// Transition to the ERROR state if applicable
IF bMyMove AND stMotionStage.bError THEN
    nState := ERROR;
    bError := TRUE;
    nErrorId := stMotionStage.nErrorId;
    bCausedError := TRUE;
END_IF
sErrorMessage := F_MotionErrorCodeLookup(nErrorId := nErrorId);

CASE nState OF
INIT, WAIT_EXEC, ERROR:
    bBusy := FALSE;
ELSE
    bBusy := TRUE;
END_CASE

END_FUNCTION_BLOCK

// POUs/Motion/States/FB_PositionStateReadND
FUNCTION_BLOCK FB_PositionStateReadND
(*
    Function block to get the combined N-dimensional state of a group of motors.
    It is a building block not meant for use outside of lcls-twintcat-motion.

    Use FB_PositionStateRead1D, FB_PositionStateRead2D, ... etc. instead
*)
VAR_IN_OUT
    // The motors with a combined N-dimensional state
    astMotionStage: ARRAY[1..MotionConstants.MAX_STATE_MOTORS] OF ST_MotionStage;
    // Each motor's respective position states along its direction
    astPositionState: ARRAY[1..MotionConstants.MAX_STATE_MOTORS] OF ARRAY[1..GeneralConstants.MAX_STATES] OF ST_PositionState;
END_VAR
VAR_INPUT
    // The number of motors we're actually using
    nActiveMotorCount: UINT;
END_VAR
VAR_OUTPUT
    // TRUE if we're standing still at a known state.
    bKnownState: BOOL;
    // TRUE if we're moving, there can be no valid state if we are moving.
    bMovingState: BOOL;
    // If we're at a known state, this will be the state index along the enclosed states arrays. Otherwise, it will be zero, which is below the bounds of the states array.
    nPositionIndex: UINT;
    // TRUE if the active motor count was invalid
    bMotorCountError: BOOL;
    // A full description of whether we're at each of our states. This is used to clarify cases where states may overlap.
    abAtPosition: ARRAY[1..GeneralConstants.MAX_STATES] OF BOOL;
END_VAR
VAR
    // The individual position state reader function blocks
    afbPositionStateRead: ARRAY[1..MotionConstants.MAX_STATE_MOTORS] OF FB_PositionStateRead;

    nIter: UINT;
    nIter2: UINT;
END_VAR


CheckCount();
IF NOT bMotorCountError THEN
    DoStateReads();
    CombineOutputs();
END_IF

ACTION CheckCount:

// Make sure the motor count is valid (positive, nonzero, less or equal to the max)
bMotorCountError S= nActiveMotorCount <= 0;
bMotorCountError S= nActiveMotorCount > MotionConstants.MAX_STATE_MOTORS;
END_ACTION

ACTION CombineOutputs:

// bKnownState is TRUE if ALL motors have the same known state
bKnownState := TRUE;
FOR nIter := 1 TO nActiveMotorCount DO
    bKnownState := bKnownState AND afbPositionStateRead[nIter].bKnownState;
END_FOR

// bMovingState is TRUE if ANY motor is moving
bMovingState := FALSE;
FOR nIter := 1 TO nActiveMotorCount DO
    bMovingState := bMovingState OR afbPositionStateRead[nIter].bMovingState;
END_FOR

// To account for redundant 1D states, we need to check the full output arrays.
nPositionIndex := 0;
FOR nIter := 1 TO GeneralConstants.MAX_STATES DO
    abAtPosition[nIter] := TRUE;
    FOR nIter2 := 1 TO nActiveMotorCount DO
        abAtPosition[nIter] R= NOT afbPositionStateRead[nIter2].abAtPosition[nIter];
    END_FOR
    IF abAtPosition[nIter] THEN
        nPositionIndex := nIter;
    END_IF
END_FOR

// Position index 0 means different positions
bKnownState := bKnownState AND nPositionIndex <> 0;
END_ACTION

ACTION DoStateReads:

MOTION_GVL.nMaxStateMotorCount := MAX(MOTION_GVL.nMaxStateMotorCount, nActiveMotorCount);
FOR nIter := 1 TO nActiveMotorCount DO
    afbPositionStateRead[nIter](
        stMotionStage:=astMotionStage[nIter],
        astPositionState:=astPositionState[nIter],
    );
END_FOR
END_ACTION

END_FUNCTION_BLOCK

// POUs/Motion/States/FB_PositionStateRead
FUNCTION_BLOCK FB_PositionStateRead
(*
    This function block tells us what state a single motor is at.
    In the case of multiple valid overlapping states, one will be picked arbitrarily,
    but we can see a full description of which overlapping states are present using the abAtPosition array.

    This will only run properly if FB_PositionStateInternal has been called on each position state to initialize it.
*)
VAR_IN_OUT
    // The motor to check the state of
    stMotionStage: ST_MotionStage;
    // The allowed states for this motor
    astPositionState: ARRAY[1..GeneralConstants.MAX_STATES] OF ST_PositionState;
END_VAR
VAR_OUTPUT
    // TRUE if we're standing still at a known state, or moving within the bounds of a state to another location in the bounds.
    bKnownState: BOOL;
    // TRUE if we're moving to some other state or to another non-state position.
    bMovingState: BOOL;
    // If we're at a known state, this will be the index in the astPositionState array that matches the state. Otherwise, this will be 0, which is below the bounds of the array, so it cannot be confused with a valid output.
    nPositionIndex: UINT;
    // A copy of the details of the current position state, for convenience. This may be a moving state or an unknown state as a placeholder if we are not at a known state.
    stCurrentPosition: ST_PositionState;
    // A full description of whether we're at each of our states. This is used in 2D, 3D, etc. to clarify cases where states may overlap in 1D.
    abAtPosition: ARRAY[1..GeneralConstants.MAX_STATES] OF BOOL;
END_VAR
VAR
    nIter: UINT;
END_VAR


bKnownState := FALSE;
bMovingState := FALSE;

FOR nIter := 1 TO GeneralConstants.MAX_STATES DO
    IF astPositionState[nIter].bValid THEN
        MOTION_GVL.nMaxStates := MAX(MOTION_GVL.nMaxStates, nIter);
    END_IF
    IF F_AtPositionState(stMotionStage:=stMotionStage, stPositionState:=astPositionState[nIter]) THEN
        bKnownState := TRUE;
        nPositionIndex := nIter;
        stCurrentPosition := astPositionState[nIter];
        abAtPosition[nIter] := TRUE;
    ELSE
        abAtPosition[nIter] := FALSE;
    END_IF
END_FOR

IF NOT bKnownState THEN
    nPositionIndex := 0;
    stCurrentPosition.fPosition := stMotionStage.stAxisStatus.fActPosition;
    stCurrentPosition.fDelta := 0;
    stCurrentPosition.bMoveOk := FALSE;
    stCurrentPosition.bValid := FALSE;
    stCurrentPosition.bUseRawCounts := FALSE;

    bMovingState := stMotionStage.bExecute;
    IF bMovingState THEN
        stCurrentPosition.sName := 'Moving';
        stCurrentPosition.fVelocity := stMotionStage.fVelocity;
        stCurrentPosition.fAccel := stMotionStage.fAcceleration;
    ELSE
        stCurrentPosition.sName := 'Unknown';
    END_IF
END_IF

END_FUNCTION_BLOCK

// POUs/Deprecated/FB_PositionStateManager
{attribute 'obsolete' := 'Use FB_PositionState1D instead'}
FUNCTION_BLOCK FB_PositionStateManager
(*
    Handles EPICS moves between multiple states for a single axis
    Should be wrapped inside a block with enums for states,
    see FB_EpicsInOut for an example.
*)
VAR_IN_OUT
    // Motor to move
    stMotionStage: ST_MotionStage;

    // Allocated space for 15 states besides Unknown (16 is the max for an EPICS MBBI)
    {attribute 'pytmc' := '
        pv:
        io: io
        expand: %.2d
    '}
    arrStates: ARRAY[1..15] OF ST_PositionState;

    // Corresponding arrStates index to move to, or 0 if no move selected
    setState: INT;
END_VAR
VAR_INPUT
    // If TRUE, start a move when setState transitions to a nonzero number
    bEnable: BOOL;
    // On rising edge, reset this FB
    {attribute 'pytmc' := '
        pv: RESET
        io: io
        field: ZNAM False
        field: ONAM True
    '}
    bReset: BOOL;
END_VAR
VAR_OUTPUT
    // If TRUE, there is an error
    {attribute 'pytmc' := '
        pv: ERR
        io: i
        field: ZNAM False
        field: ONAM True
    '}
    bError: BOOL;
    // Error ID
    {attribute 'pytmc' := '
        pv: ERRID
        io: i
    '}
    nErrorId: UDINT;
    // The error that caused bError to flip TRUE
    {attribute 'pytmc' := '
        pv: ERRMSG
        io: i
    '}
    sErrorMessage: STRING;
    // If TRUE, we are moving the motor
    {attribute 'pytmc' := '
        pv: BUSY
        io: i
        field: ZNAM False
        field: ONAM True
    '}
    bBusy: BOOL;
    // If TRUE, we are not moving the motor and the last move completed successfully
    {attribute 'pytmc' := '
        pv: DONE
        io: i
        field: ZNAM False
        field: ONAM True
    '}
    bDone: BOOL;

    // The current position we are trying to reach, or 0
    goalState: INT;
    // The readback position
    getState: INT;
END_VAR
VAR
    bInit: BOOL;
    stUnknown: ST_PositionState;
    stGoal: ST_PositionState;
    fbStateMove: FB_PositionStateMove;
    fbStateInternal: ARRAY[1..15] OF FB_PositionStateInternal;
    nIndex: INT;
    bNewGoal: BOOL;
    bInnerExec: BOOL;
    bInnerReset: BOOL;
    rtReset: R_TRIG;
    bMoveRequested: BOOL;
END_VAR

// Reset just goes through the first-cycle init again
rtReset(CLK:=bReset);
IF rtReset.Q THEN
    bInit := FALSE;
END_IF

// First-cycle init
IF NOT bInit THEN
    bError := FALSE;
    sErrorMessage := '';
    bBusy := FALSE;
    bDone := FALSE;
    bNewGoal := FALSE;
    bInnerExec := FALSE;
    bInnerReset := TRUE;
    setState := 0;
    goalState := 0;
END_IF

// All state internal handlers
FOR nIndex := 1 TO 15 DO
    IF arrStates[nIndex].bValid THEN
        fbStateInternal[nIndex](
            stMotionStage:=stMotionStage,
            stPositionState:=arrStates[nIndex]);
    END_IF
END_FOR

// Check where we are by going through all possible states.
// Note this favors the highest-number state that we're at, it's up to you to make your states mutually exclusive.
getState := 0;
FOR nIndex := 1 TO 15 DO
    IF F_AtPositionState(stMotionStage:=stMotionStage, stPositionState:=arrStates[nIndex]) THEN
        getState := nIndex;
    END_IF
END_FOR

// Use the changing set pv as a rising-edge trigger
IF setState <> goalState THEN
    goalState := setState;
    bNewGoal := TRUE;
END_IF

// Special move handling for error/enable state
IF bError OR NOT bEnable THEN
    bInnerExec := FALSE;
// Reset inner block this cycle if we were already moving but want a new move
ELSIF bInnerExec AND bNewGoal THEN
    bInnerExec := FALSE;
    bInnerReset := TRUE;
// If we hit this branch, we're starting a new move
ELSIF bNewGoal THEN
    bInnerExec := TRUE;
    bInnerReset := FALSE;
    bNewGoal := FALSE;
END_IF

// Pick the correct goal structure or Unknown
IF goalState = 0 THEN
    stGoal := stUnknown;
ELSE
    stGoal := arrStates[goalState];
END_IF

// Do the move
fbStateMove(
    stMotionStage := stMotionStage,
    stPositionState := stGoal,
    bExecute := bInnerExec,
    bReset := bInnerReset,
    enumMotionRequest := E_MotionRequest.INTERRUPT,
    bBusy => bBusy);

// Only pass up bDone information if this FB is active
IF bInnerExec THEN
    bDone := fbStateMove.bDone;
END_IF

// Pick up any new errors, but don't override uncleared existing errors
IF NOT bError THEN
    bError := fbStateMove.bError;
    nErrorId := fbStateMove.nErrorId;
    sErrorMessage := fbStateMove.sErrorMessage;
END_IF

// Reset the setpoint and goal to 0 if we're not doing anything
// because FB is waiting for a change from 0 to "something"
bMoveRequested := bInnerExec AND NOT bDone;
IF NOT bError AND NOT bNewGoal AND NOT bMoveRequested THEN
    setState := 0;
    goalState := 0;
    bInnerExec := FALSE;
END_IF

// Bring inner reset back low at the end of the init cycle so that it can be triggered again later
IF NOT bInit THEN
    bInit := TRUE;
    bInnerReset := FALSE;
END_IF

END_FUNCTION_BLOCK

// POUs/Deprecated/FB_PositionStateBase
{attribute 'obsolete' := 'Use FB_PositionState1D instead'}
FUNCTION_BLOCK FB_PositionStateBase
(*
    Handles EPICS moves between multiple states for a single axis
    Should be subclassed for a specific enumSet and enumGet.
    See body comment  or FB_PositionStateInOut for an implementation example.
*)
VAR_IN_OUT
    // Motor to move
    stMotionStage: ST_MotionStage;
END_VAR
VAR_INPUT
    // If TRUE, start a move when setState transitions to a nonzero number
    bEnable: BOOL;
    // On rising edge, reset this FB
    {attribute 'pytmc' := '
        pv: RESET
        io: io
        field: ZNAM False
        field: ONAM True
    '}
    bReset: BOOL;
END_VAR
VAR_OUTPUT
    // If TRUE, there is an error
    {attribute 'pytmc' := '
        pv: ERR
        io: i
        field: ZNAM False
        field: ONAM True
    '}
    bError: BOOL;
    // Error ID
    {attribute 'pytmc' := '
        pv: ERRID
        io: i
    '}
    nErrorId: UDINT;
    // The error that caused bError to flip TRUE
    {attribute 'pytmc' := '
        pv: ERRMSG
        io: i
    '}
    sErrorMessage: STRING;
    // If TRUE, we are moving the motor
    {attribute 'pytmc' := '
        pv: BUSY
        io: i
        field: ZNAM False
        field: ONAM True
    '}
    bBusy: BOOL;
    // If TRUE, we are not moving the motor and the last move completed successfully
    {attribute 'pytmc' := '
        pv: DONE
        io: i
        field: ZNAM False
        field: ONAM True
    '}
    bDone: BOOL;
END_VAR
VAR
    // Pre-allocated array of states
    {attribute 'pytmc' := '
        pv:
        io: io
        expand: %.2d
    '}
    arrStates: ARRAY[1..GeneralConstants.MAX_STATES] OF ST_PositionState;

    // Corresponding arrStates index to move to, or 0 if no move selected
    setState: INT;
    // The current position we are trying to reach, or 0
    goalState: INT;
    // The readback position
    getState: INT;

    bInit: BOOL;
    stUnknown: ST_PositionState;
    stGoal: ST_PositionState;
    fbStateMove: FB_PositionStateMove;
    fbStateInternal: ARRAY[1..GeneralConstants.MAX_STATES] OF FB_PositionStateInternal;
    nIndex: INT;
    bNewGoal: BOOL;
    bInnerExec: BOOL;
    bInnerReset: BOOL;
    rtReset: R_TRIG;
    bMoveRequested: BOOL;
END_VAR

(*
    Subclass me, define enums to translate setState and getState, call Exec

    Example:

    <something to fill arrStates>
    setState := enumSet;
    Exec();
    enumGet := getState;
    enumSet := setState;
*)

ACTION Exec:
StateHandler();
END_ACTION

ACTION StateHandler:
// Reset just goes through the first-cycle init again
rtReset(CLK:=bReset);
IF rtReset.Q THEN
    bInit := FALSE;
    bReset := FALSE;
END_IF

// First-cycle init
IF NOT bInit THEN
    bError := FALSE;
    nErrorID := 0;
    sErrorMessage := '';
    bBusy := FALSE;
    bDone := FALSE;
    bNewGoal := FALSE;
    bInnerExec := FALSE;
    bInnerReset := TRUE;
    setState := 0;
    goalState := 0;
END_IF

// All state internal handlers
FOR nIndex := 1 TO GeneralConstants.MAX_STATES DO
    IF arrStates[nIndex].bValid THEN
        fbStateInternal[nIndex](
            stMotionStage:=stMotionStage,
            stPositionState:=arrStates[nIndex]);
    END_IF
END_FOR

// Check where we are by going through all possible states.
// Note this favors the highest-number state that we're at, it's up to you to make your states mutually exclusive.
getState := 0;
FOR nIndex := 1 TO GeneralConstants.MAX_STATES DO
    IF F_AtPositionState(stMotionStage:=stMotionStage, stPositionState:=arrStates[nIndex]) THEN
        getState := nIndex;
    END_IF
END_FOR

// Use the changing set pv as a rising-edge trigger
IF setState <> goalState THEN
    goalState := setState;
    bNewGoal := TRUE;
END_IF

// Special move handling for error/enable state
IF bError OR NOT bEnable THEN
    bInnerExec := FALSE;
ELSIF bNewGoal THEN
    IF fbStateMove.bBusy THEN
        // Stop previous move if we were already moving but want a new move
        bInnerExec := FALSE;
    ELSE
        // If we hit this branch, we're ready to start a new move
        bInnerExec := TRUE;
        bInnerReset := FALSE;
        bNewGoal := FALSE;
    END_IF
END_IF

// Pick the correct goal structure or Unknown
IF goalState = 0 THEN
    stGoal := stUnknown;
ELSE
    stGoal := arrStates[goalState];
END_IF

// Do the move
fbStateMove(
    stMotionStage := stMotionStage,
    stPositionState := stGoal,
    bExecute := bInnerExec,
    bReset := bInnerReset,
    enumMotionRequest := E_MotionRequest.INTERRUPT,
    bBusy => bBusy);

// Only pass up bDone information if this FB is active
IF bInnerExec THEN
    bDone := fbStateMove.bDone;
END_IF

// Pick up any new errors, but don't override uncleared existing errors
IF NOT bError THEN
    bError := fbStateMove.bError;
    IF bError THEN
        nErrorId := fbStateMove.nErrorId;
        sErrorMessage := fbStateMove.sErrorMessage;
    END_IF
END_IF

// Reset the setpoint and goal to 0 if we're not doing anything
// because FB is waiting for a change from 0 to "something"
bMoveRequested := bInnerExec AND NOT bDone;
IF NOT bError AND NOT bNewGoal AND NOT bMoveRequested THEN
    setState := 0;
    goalState := 0;
    bInnerExec := FALSE;
END_IF

// Bring inner reset back low at the end of the init cycle so that it can be triggered again later
IF NOT bInit THEN
    bInit := TRUE;
    bInnerReset := FALSE;
END_IF
END_ACTION

END_FUNCTION_BLOCK

// POUs/Deprecated/FB_PositionStateInOut
{attribute 'obsolete' := 'Use FB_PositionState1D_InOut instead'}
FUNCTION_BLOCK FB_PositionStateInOut EXTENDS FB_PositionStateBase
(*
    Example usage of FB_PositionStateBase for a simple IN/OUT axis. See NOTE: comments.
    Also usable as a drop-in for these cases (no need to roll your own in/out)
*)
VAR_INPUT
    // The enum position to move to
    {attribute 'pytmc' := '
        pv: SET
        io: io
    '}
    enumSet: ENUM_EpicsInOut_INT; // NOTE: Please copy this pragma exactly on your enumSet

    // Information about the OUT position
    stOut: ST_PositionState; // NOTE: Do not pragma these, let it happen in the manager.
    // Information about the IN position
    stIn: ST_PositionState;
END_VAR
VAR_OUTPUT
    // The enum state readback
    {attribute 'pytmc' := '
        pv: GET
        io: i
    '}
    enumGet: ENUM_EpicsInOut_INT; // NOTE: Please copy this pragma exactly on your enumGet
END_VAR
VAR
    bInOutInit: BOOL;
END_VAR

IF NOT bInOutInit THEN
    bInOutInit := TRUE;
    arrStates[1] := stOut;
    arrStates[2] := stIn;
    stOut.sName := 'OUT';
    stIn.sName := 'IN';
END_IF
setState := enumSet;
Exec();
enumGet := getState;
enumSet := setState;

END_FUNCTION_BLOCK

// POUs/Deprecated/FB_PositionStateBase_WithPMPS
{attribute 'obsolete' := 'Use FB_PositionStatePMPS1D instead'}
FUNCTION_BLOCK FB_PositionStateBase_WithPMPS EXTENDS FB_PositionStateBase
(*
    Handles EPICS moves between multiple states for a single axis with PMPS.
    Should be subclassed for a specific enumSet and enumGet.
    See body comment  or FB_PositionStateInOut_WithPMPS for an implementation example.
*)
VAR_IN_OUT
    fbArbiter: FB_Arbiter;
    fbFFHWO: FB_HardwareFFOutput;
END_VAR
VAR_INPUT
    sPmpsDeviceName: STRING;
    sTransitionKey: STRING;
    {attribute 'pytmc' := '
        pv: PMPS:ARB:ENABLE
        io: io
    '}
    bArbiterEnabled: BOOL := TRUE;
    tArbiterTimeout: TIME := T#1s;
    bMoveOnArbiterTimeout: BOOL := TRUE;
    fStateBoundaryDeadband: LREAL := 0;
    bBPOKAutoReset: BOOL := False;
END_VAR
VAR
    {attribute 'pytmc' := 'pv: PMPS'}
    fbStatePMPS: FB_PositionStatePMPS;
    fbEncErrFFO: FB_EncErrorFFO;
END_VAR

(*
    Subclass me, define enums to translate setState and getState, call Exec

    Example:

    <something to fill arrStates>
    setState := enumSet;
    Exec();
    enumGet := getState;
    enumSet := setState;
*)

ACTION Exec:
StateHandler();
PMPSHandler();
END_ACTION

ACTION PMPSHandler:
fbStatePMPS(
    fbArbiter:=fbArbiter,
    fbFFHWO:=fbFFHWO,
    stMotionStage:=stMotionStage,
    arrStates:=arrStates,
    sPmpsDeviceName:=sPmpsDeviceName,
    sTransitionKey:=sTransitionKey,
    stPmpsDoc:= PMPS_GVL.BP_jsonDoc,
    bRequestTransition:=setState <> 0,
    setState:=setState,
    getState:=getState,
    bArbiterEnabled:=bArbiterEnabled,
    tArbiterTimeout:=tArbiterTimeout,
    bMoveOnArbiterTimeout:=bMoveOnArbiterTimeout,
    fStateBoundaryDeadband:=fStateBoundaryDeadband,
    bBPOKAutoReset:=bBPOKAutoReset);

fbEncErrFFO(
    stMotionStage:=stMotionStage,
    fbFFHWO:=fbFFHWO,
    bAutoReset:=TRUE);
END_ACTION

END_FUNCTION_BLOCK

// POUs/Deprecated/FB_PositionStateInOut_WithPMPS
{attribute 'obsolete' := 'Use FB_PositionStatePMPS1D_InOut instead'}
FUNCTION_BLOCK FB_PositionStateInOut_WithPMPS EXTENDS FB_PositionStateBase_WithPMPS
(*
    Example usage of FB_PositionStateBase_WithPMPS for a simple IN/OUT axis. See NOTE: comments.
    Also usable as a drop-in for these cases (no need to roll your own in/out)

    This is the PMPS version. Note that the only difference is that we extend the _WithPMPS FB.
*)
VAR_INPUT
    // The enum position to move to
    {attribute 'pytmc' := '
        pv: SET
        io: io
    '}
    enumSet: ENUM_EpicsInOut_INT; // NOTE: Please copy this pragma exactly on your enumSet

    // Information about the OUT position
    stOut: ST_PositionState; // NOTE: Do not pragma these, let it happen in the manager.
    // Information about the IN position
    stIn: ST_PositionState;
END_VAR
VAR_OUTPUT
    // The enum state readback
    {attribute 'pytmc' := '
        pv: GET
        io: i
    '}
    enumGet: ENUM_EpicsInOut_INT; // NOTE: Please copy this pragma exactly on your enumGet
END_VAR
VAR
    bInOutInit: BOOL;
END_VAR

IF NOT bInOutInit THEN
    bInOutInit := TRUE;
    arrStates[1] := stOut;
    arrStates[2] := stIn;
    stOut.sName := 'OUT';
    stIn.sName := 'IN';
END_IF
setState := enumSet;
Exec();
enumGet := getState;
enumSet := setState;

END_FUNCTION_BLOCK

// POUs/Motion/States/Examples/FB_PositionStatePMPS1D_InOut
FUNCTION_BLOCK FB_PositionStatePMPS1D_InOut
(*
    An example and usable drop-in instance for a 1D pmps state device with just an IN and an OUT state.
    Note that the outward-facing API is nearly identical to the non-PMPS version
*)
VAR_IN_OUT
    // Include a stage that can be passed into the FB
    stMotionStage: ST_MotionStage;
    // Simplify the interface, the user just needs to construct and pass in and out position states
    stIn: ST_PositionState;
    stOut: ST_PositionState;
    // Include PMPS output helpers
    fbFFHWO: FB_HardwareFFOutput;
    fbArbiter: FB_Arbiter;
END_VAR
VAR_INPUT
    // Define an ENUM for EPICS to use to set a new value. It is expected this will be written to during one cycle, so don't continually apply a value here in the PLC code.
    // It is exposed as an input so we can test it using the PLC.
    {attribute 'pytmc' := '
      pv: STATE:SET
      io: io
    '}
    eStateSet: E_EpicsInOut;
END_VAR
VAR_OUTPUT
    // Define an ENUM for EPICS to use to report the new value.
    {attribute 'pytmc' := '
      pv: STATE:GET
      io: i
    '}
    eStateGet: E_EpicsInOut;
END_VAR
VAR
    // Include the standard fb with blank pv pragma
    {attribute 'pytmc' := 'pv:'}
    fbPositionStatePMPS1D: FB_PositionStatePMPS1D;
    // The standard fb expects a full array of position states
    astPositionState: ARRAY[1..GeneralConstants.MAX_STATES] OF ST_PositionState;
END_VAR


// Optional: default state names
IF stIn.sName = '' THEN
    stIn.sName := 'IN';
END_IF
IF stOut.sName = '' THEN
    stOut.sName := 'OUT';
END_IF

// Assemble the states array, matching the enum values
astPositionState[E_EpicsInOut.OUT] := stOut;
astPositionState[E_EpicsInOut.IN] := stIn;

// Call the main function block, passing our motors, states, and an enable
fbPositionStatePMPS1D(
    fbFFHWO:=fbFFHWO,
    fbArbiter:=fbArbiter,
    stMotionStage:=stMotionStage,
    astPositionState:=astPositionState,
    eEnumSet:=eStateSet,
    eEnumGet:=eStateGet,
    bEnableMotion:=TRUE,
    bEnableBeamParams:=TRUE,
    bEnablePositionLimits:=TRUE,
);

// Send updates made on the array back to the inputs (VAR_IN_OUT) for maximum clarity
stOut := astPositionState[E_EpicsInOut.OUT];
stIn := astPositionState[E_EpicsInOut.IN];

END_FUNCTION_BLOCK

// POUs/Deprecated/FB_PositionStatePMPS
{attribute 'obsolete' := 'Use FB_PositionStatePMPS1D instead'}
FUNCTION_BLOCK FB_PositionStatePMPS EXTENDS FB_PositionStatePMPS_Base
(*
    Hooks up a position state to an arbiter and an FFO
        Use BeamParameterTransitionManager to manage transition requests between states
        Hook up to the inputs/outputs of the state function block
        Raises FFO if beam parameters are worse than required for current state
*)
VAR_IN_OUT
    fbArbiter: FB_Arbiter;
    fbFFHWO: FB_HardwareFFOutput;
END_VAR
VAR_INPUT
    bReadPmpsDb: BOOL;
    sPmpsDeviceName: STRING;
    sTransitionKey: STRING;
    stPmpsDoc: SJsonValue;
    stHighBeamThreshold: ST_BeamParams := PMPS_GVL.cstFullBeam;
    bBPOKAutoReset: BOOL := False;
END_VAR
VAR
    arrPMPS: ARRAY[0..GeneralConstants.MAX_STATES] OF ST_DbStateParams;
    nBPIndex: UINT;
    nTransitionAssertionID: UDINT;
    nLastReqAssertionID: UDINT;
    fbReadPmpsDb: FB_JsonDocToSafeBP;
    ftDbBusy: F_TRIG;
    rtReadDBExec: R_TRIG;
    ftRead: F_TRIG;
    bptm: BeamParameterTransitionManager;
    ffBeamParamsOk: FB_FastFault;
    ffZeroRate: FB_FastFault;
    ffBPTMTimeoutAndMove: FB_FastFault;
    ffBPTMError: FB_FastFault;
    ffMaint: FB_FastFault;
    ffUnknown: FB_FastFault;
    bFFOxOk: BOOL;
    bAtSafeState: BOOL;
    nIter: UINT;
END_VAR

Exec();

ACTION AssertHere:
fbArbiter.AddRequest(
    sDevName := stMotionStage.sName,
    nReqID := stStateReq.stPMPS.nRequestAssertionID,
    stReqBP := stStateReq.stPMPS.stBeamParams);
END_ACTION

ACTION ClearAsserts:
fbArbiter.RemoveRequest(nTransitionAssertionID);
FOR nIter := 1 TO GeneralConstants.MAX_STATES DO
    fbArbiter.RemoveRequest(arrStates[nIter].stPMPS.nRequestAssertionID);
END_FOR
END_ACTION

ACTION HandleBPTM:
(*
  Handle finishing the bptm late if timed out
  bptm needs a rising edge of bTransDone after authorizing transition
  If we fall into this block, bTransDone would otherwise be stuck at TRUE forever
  so the BPTM would never see a rising edge and therefore stay stuck
  We set to FALSE here to reset the BPTM, then gets set to TRUE again if really done.
*)
rtDoLateFinish(CLK:=bLateFinish AND bInternalAuth);
IF rtDoLateFinish.Q THEN
    bTransDone := FALSE;
    bLateFinish := FALSE;
END_IF

IF stStateReq.stPMPS.nRequestAssertionID <> nTransitionAssertionID THEN
    (*
        Edge case: the request is swapped out without a move
        Same as above: we need a rising edge of bTransDone, so cause a falling edge and the let the rising edge happen next cycle
        This will already be false when we request a positional move
    *)
    bTransDone R= stStateReq.stPMPS.nRequestAssertionID <> nLastReqAssertionID;
    // Just normal bptm call
    bptm(fbArbiter:=fbArbiter,
         i_sDeviceName:=stMotionStage.sName,
         i_TransitionAssertionID:=nTransitionAssertionID,
         i_stTransitionAssertion:=stTransitionBeam,
         i_nRequestedAssertionID:=stStateReq.stPMPS.nRequestAssertionID,
         i_stRequestedAssertion:=stStateReq.stPMPS.stBeamParams,
         i_xDoneMoving:=bTransDone,
         stCurrentBeamParameters:=PMPS_GVL.stCurrentBeamParameters,
         q_xTransitionAuthorized=>bInternalAuth,
         bDone=>bBPTMDone);
    nLastReqAssertionID := stStateReq.stPMPS.nRequestAssertionID;
END_IF
END_ACTION

ACTION HandleFFO:
// stBeamNeeded will point to Unknown/No beam if we are out of state bounds or in motion
// Otherwise we'll have the current state's beam parameters

// Check for bad conditions
bFFOxOk := F_SafeBPCompare(PMPS_GVL.stCurrentBeamParameters, stBeamNeeded);
// It is safe to reset automatically if our current state can take full beam.
// Otherwise we'll have to ask for a user acknowledgement to clear.
// This avoids rapidly cycling the FFOs on/off
// You can pass in a different stHighBeamThreshold as an input parameter to customize this behavior
bAtSafeState := F_SafeBPCompare(stHighBeamThreshold, stBeamNeeded);

// If the beam parameters are wrong, it is a fault! This encompasses all unknown arbiter-related errors.
ffBeamParamsOk.i_xOK := bFFOxOk;
ffBeamParamsOk.i_xReset S= bFFOxOk AND bAtSafeState;
ffBeamParamsOk.i_xReset R= NOT ffBeamParamsOk.i_xOK;
ffBeamParamsOk.i_xAutoReset := bBPOKAutoReset;

ffBeamParamsOk(
    i_DevName:=stMotionStage.sName,
    i_Desc:='Beam parameter mismatch',
    i_TypeCode:=16#1000,
    io_fbFFHWO:=fbFFHWO);

// Trip the beam for zero-rate states. This is a PMPS training wheel and should ultimately be removed.
// Note: I think this is already redundant
ffZeroRate(
    i_xOk := stBeamNeeded.nRate > 0,
    i_xAutoReset := TRUE,
    i_DevName := stMotionStage.sName,
    i_Desc := 'Device requesting zero rate',
    i_TypeCode := 16#1001,
    io_fbFFHWO := fbFFHWO);

// Trip the beam for BPTM timeouts if we want to move
// Only reset at safe beam OR at no bptm errors (some other FF should catch additional issues)
ffBPTMTimeoutAndMove.i_xOK := NOT (bArbiterTimeout AND bMoveOnArbiterTimeout);
ffBPTMTimeoutAndMove.i_xReset S= bAtSafeState OR (bptm.bDone AND NOT bptm.bError);
ffBPTMTimeoutAndMove.i_xReset R= NOT ffBPTMTimeoutAndMove.i_xOK;
ffBPTMTimeoutAndMove(
    i_DevName := stMotionStage.sName,
    i_Desc := 'BPTM Timeout',
    i_TypeCode := 16#1002,
    io_fbFFHWO := fbFFHWO);

// Trip the beam for BPTM Errors
ffBPTMError.i_xOK := NOT bptm.bError;
ffBPTMError.i_xReset S= bptm.bDone AND NOT bptm.bError;
ffBPTMError.i_xReset R= NOT ffBPTMError.i_xOK;
ffBPTMError(
    i_DevName := stMotionStage.sName,
    i_Desc := 'BPTM error, state transition failed',
    i_TypeCode := 16#1003,
    io_fbFFHWO := fbFFHWO);

// Trip the beam for maintenance mode
ffMaint(
    i_xOK := NOT bMaintMode,
    i_xAutoReset := TRUE,
    i_DevName := stMotionStage.sName,
    i_Desc := 'Device is in maintenance mode',
    i_TypeCode := 16#1004,
    io_fbFFHWO := fbFFHWO);

// Trip the beam for unknown state
ffUnknown(
    i_xOK := getState > 0 OR bInTransition,
    i_xAutoReset := TRUE,
    i_DevName := stMotionStage.sName,
    i_Desc := 'Unknown position between moves',
    i_TypeCode := 16#1005,
    io_fbFFHWO := fbFFHWO);
END_ACTION

ACTION HandlePmpsDb:

// Automatically read from the pmps db when it updates
// Assume update if no longer busy and no errors

ftDbBusy(CLK:=MOTION_GVL.fbPmpsFileReader.bBusy);
IF ftDbBusy.Q THEN
    bReadPmpsDb S= NOT MOTION_GVL.fbPmpsFileReader.bError;
END_IF

rtReadDBExec(CLK:=bReadPmpsDb);
IF rtReadDBExec.Q THEN
    arrPMPS[0].sPmpsState := sTransitionKey;
    FOR nBPIndex := 1 TO GeneralConstants.MAX_STATES BY 1 DO
        arrPMPS[nBPIndex] := arrStates[nBPIndex].stPMPS;
    END_FOR
END_IF

fbReadPmpsDb(
    bExecute:=bReadPmpsDb,
    jsonDoc:=stPmpsDoc,
    sDeviceName:=sPmpsDeviceName,
    io_fbFFHWO:=fbFFHWO,
    arrStates:=arrPMPS,
);
bReadPmpsDb R= NOT fbReadPmpsDb.bBusy;

ftRead(CLK:=fbReadPmpsDb.bBusy);

stTransitionState.sName := 'Transition';
IF ftRead.Q AND NOT fbReadPmpsDb.bError THEN
    stTransitionDb := arrPMPS[0];
    stTransitionBeam := arrPMPS[0].stBeamParams;
    nTransitionAssertionID := arrPMPS[0].nRequestAssertionID;
    stTransitionState.stPMPS := arrPMPS[0];
    FOR nBPIndex := 1 TO GeneralConstants.MAX_STATES BY 1 DO
        arrStates[nBPIndex].stPMPS := arrPMPS[nBPIndex];
    END_FOR
END_IF
END_ACTION

END_FUNCTION_BLOCK

// POUs/Deprecated/FB_PositionStatePMPS_Base
{attribute 'obsolete' := 'Use FB_PositionStatePMPS1D instead'}
FUNCTION_BLOCK FB_PositionStatePMPS_Base
(*
    FB_PositionStatePMPS without Arbiter, BPTM, FFO

    This allows me to test most of the code without an arbiter plc setup
*)
VAR_IN_OUT
    stMotionStage: ST_MotionStage;
    arrStates: ARRAY[1..GeneralConstants.MAX_STATES] OF ST_PositionState;
END_VAR
VAR_INPUT
    bArbiterEnabled: BOOL := TRUE;
    {attribute 'pytmc' := '
        pv: MAINT
        io: io
    '}
    bMaintMode: BOOL;
    bRequestTransition: BOOL;
    setState: INT;
    getState: INT;
    fStateBoundaryDeadband: LREAL := 0;
    tArbiterTimeout: TIME := T#1s;
    bMoveOnArbiterTimeout: BOOL := TRUE;
END_VAR
VAR_OUTPUT
    bTransitionAuthorized: BOOL;
    bForwardAuthorized: BOOL;
    bBackwardAuthorized: BOOL;
    bArbiterTimeout: BOOL;
END_VAR
VAR
    {attribute 'pytmc' := '
        pv: TRANS
        io: i
    '}
    stTransitionDb: ST_DbStateParams;
    stTransitionBeam: ST_BeamParams := PMPS_GVL.cst0RateBeam;
    stTransitionState: ST_PositionState;
    bInit: BOOL := TRUE;
    bTransDone: BOOL;
    rtTransReq: R_TRIG;
    bBPTMDone: BOOL;
    rtBPTMDone: R_TRIG;
    ftMotorExec: F_TRIG;
    rtTransDone: R_TRIG;
    rtDoLateFinish: R_TRIG;
    tonDone: TON;
    stStateReq: ST_PositionState;
    mcPower: MC_POWER;
    fUpperBound: LREAL;
    fLowerBound: LREAL;
    nGoalState: INT;
    stGoalState: ST_PositionState;
    fActPos: LREAL;
    fReqPos: LREAL;
    bInTransition: BOOL;
    stBeamNeeded: ST_BeamParams;
    bFwdOk: BOOL;
    bBwdOk: BOOL;
    tonArbiter: TON;
    bLateFinish: BOOL;
    bInternalAuth: BOOL;
END_VAR

// This is meant to be subclassed. The parent class body is in the Exec action.

ACTION AssertHere:

END_ACTION

ACTION ClearAsserts:

END_ACTION

ACTION Exec:

// Load the pmps parameters as needed
HandlePmpsDb();

// Initialize or reinitialize to the current state value
rtBPTMDone(CLK:=bBPTMDone);
ftMotorExec(CLK:=stMotionStage.bExecute);
tonDone(
    IN:=bTransDone,
    PT:=T#100ms
    );
IF rtBPTMDone.Q OR ftMotorExec.Q OR tonDone.Q THEN
    bInit := TRUE;
END_IF
IF bInit OR nGoalState = 0 OR stMotionStage.bError THEN
    bInit R= stMotionStage.bAxisParamsInit;
    nGoalState := getState;
    stStateReq := GetStateStruct(getState);
    bInTransition := FALSE;
    rtTransReq(CLK:=FALSE);
    bTransitionAuthorized := FALSE;
    bArbiterTimeout := FALSE;
END_IF

// Request transition on rising edge
rtTransReq(CLK:=bRequestTransition);
IF rtTransReq.Q THEN
    nGoalState := setState;
    stStateReq := GetStateStruct(setState);
    bInTransition := TRUE;
    bTransDone := FALSE;
ELSE
    bTransDone := F_AtPositionState(stMotionStage:=stMotionStage, stPositionState:=stStateReq) AND NOT stMotionStage.bBusy;
END_IF

// Mark late finish if bTransDone -> true before the bptm is done
// This means that we finished the move so fast that the bptm needs to be unstuck via toggling bTransDone
rtTransDone(CLK:=bTransDone);
bLateFinish S= rtTransDone.Q AND NOT bBPTMDone;

IF bArbiterEnabled THEN
    // Handles getting the request to the arbiter and back
    HandleBPTM();
    // Handle arbiter timeouts
    IF tArbiterTimeout > T#0s THEN
        tonArbiter(
            IN:=bInTransition AND NOT bInternalAuth,
            PT:=tArbiterTimeout,
            Q=>bArbiterTimeout);
    ELSE
        bArbiterTimeout := FALSE;
    END_IF
    bTransitionAuthorized S= bInternalAuth OR (bArbiterTimeout AND bMoveOnArbiterTimeout);
ELSE
    // Clear all of our assertions if we decide to disable the arbiter
    ClearAsserts();
    // Do some dummy request handling
    bTransitionAuthorized := stMotionStage.bExecute;
    bArbiterTimeout := stMotionStage.bExecute;
END_IF

// Set up MPS virtual limit for moves at and between states
stGoalState := GetStateStruct(nGoalState);
fActPos := stMotionStage.stAxisStatus.fActPosition;
IF stMotionStage.bExecute THEN
    fReqPos := stMotionStage.fPosition;
ELSE
    fReqPos := fActPos;
END_IF

// Start with no move authority
bForwardAuthorized := FALSE;
bBackwardAuthorized := FALSE;

// Check if it would be OK to move without granting auth
bFwdOk := F_PosUnderUpperBound(MAX(fActPos, fReqPos) + ABS(fStateBoundaryDeadband), stGoalState);
bBwdOk := F_PosOverLowerBound(MIN(fActPos, fReqPos) - ABS(fStateBoundaryDeadband), stGoalState);

// Grant auth during moves based on goal state, current position, and goal position
IF stMotionStage.bExecute AND stGoalState.bValid THEN
    bForwardAuthorized := bFwdOk;
    bBackwardAuthorized := bBwdOk;
END_IF

IF bInTransition THEN
    // Deny auth during a transition request until transition is authorized
    bForwardAuthorized R= NOT bTransitionAuthorized;
    bBackwardAuthorized R= NOT bTransitionAuthorized;
    // Have the motor wait for permission to start move instead of immediately erroring
    stMotionStage.bSafetyReady := bTransitionAuthorized;
ELSE
    // If not transitioning, no need to wait for safety: immediately try to move and error if no auth
    stMotionStage.bSafetyReady := stMotionStage.bExecute;
    // Set an error message override in case this causes an error
    IF stMotionStage.bError AND bArbiterEnabled AND NOT bMaintMode THEN
        IF fReqPos > fActPos AND NOT bFwdOk THEN
            stMotionStage.sCustomErrorMessage := 'Unsafe tweak forward blocked by PMPS';
        ELSIF fReqPos < fActPos AND NOT bBwdOk THEN
            stMotionStage.sCustomErrorMessage := 'Unsafe tweak backward blocked by PMPS';
        END_IF
    END_IF
END_IF

IF bArbiterEnabled AND NOT bMaintMode THEN
// Only let us move if the transition is allowed, or if we are moving within a state's bounds
    mcPower(Axis:=stMotionStage.Axis,
            Enable:=stMotionStage.bAllEnable,
            Enable_Positive:=stMotionStage.bAllForwardEnable AND bForwardAuthorized,
            Enable_Negative:=stMotionStage.bAllBackwardEnable AND bBackwardAuthorized);
ELSE
    mcPower(Axis:=stMotionStage.Axis,
            Enable:=stMotionStage.bAllEnable,
            Enable_Positive:=stMotionStage.bAllForwardEnable,
            Enable_Negative:=stMotionStage.bAllBackwardEnable);
    stMotionStage.bSafetyReady := TRUE;
END_IF

// Raise fast faults as needed
stBeamNeeded := GetBeamFromState(getState);
HandleFFO();
END_ACTION

METHOD GetBeamFromState : ST_BeamParams;
VAR_INPUT
    nState: INT;
END_VAR
VAR
    stState: ST_PositionState;
END_VAR
stState := GetStateStruct(nState);
GetBeamFromState := stState.stPMPS.stBeamParams;
END_METHOD

METHOD GetStateCode : INT
VAR_INPUT
    nState: INT;
END_VAR
IF nState < 0 OR nState > GeneralConstants.MAX_STATES THEN
    GetStateCode := -1;
ELSE
    GetStateCode := nState;
END_IF
END_METHOD

METHOD GetStateStruct : ST_PositionState
VAR_INPUT
    nState: INT;
END_VAR
{warning disable C0371}
// Implicit VAR_IN_OUT reference inside a method needs special handling
IF NOT __ISVALIDREF(arrStates) THEN
    GetStateStruct := stTransitionState;
    RETURN;
END_IF
CASE GetStateCode(nState) OF
    -1: GetStateStruct := stTransitionState;
    0: GetStateStruct := stTransitionState;
    ELSE
        GetStateStruct := arrStates[nState];
END_CASE
{warning restore C0371}
END_METHOD

ACTION HandleBPTM:

END_ACTION

ACTION HandleFFO:

END_ACTION

ACTION HandlePmpsDb:

END_ACTION

END_FUNCTION_BLOCK

// POUs/Deprecated/FB_PositionStateBase_WithPMPS_Test
{attribute 'obsolete' := 'No longer any reason to use this, all state classes can have unit tests.'}
FUNCTION_BLOCK FB_PositionStateBase_WithPMPS_Test EXTENDS FB_PositionStateBase
(*
    Handles EPICS moves between multiple states for a single axis with fake PMPS.
    Should be subclassed for a specific enumSet and enumGet.
    See body comment  or FB_PositionStateInOut_WithPMPS_Test for an implementation example.
*)
VAR_INPUT
    stTransitionBeam: ST_BeamParams := PMPS_GVL.cst0RateBeam;
    nTransitionAssertionID: UDINT;
END_VAR
VAR
    fbStatePMPS: FB_PositionStatePMPS_Test;
END_VAR

(*
    Subclass me, define enums to translate setState and getState, call Exec

    Example:

    <something to fill arrStates>
    setState := enumSet;
    Exec();
    enumGet := getState;
    enumSet := setState;
*)

ACTION Exec:
StateHandler();
PMPSHandler();
END_ACTION

ACTION PMPSHandler:
fbStatePMPS(
    stMotionStage:=stMotionStage,
    arrStates:=arrStates,
    bRequestTransition:=setState <> 0,
    setState:=setState,
    getState:=getState);
END_ACTION

END_FUNCTION_BLOCK

// POUs/Deprecated/FB_PositionStateInOut_WithPMPS_Test
{attribute 'obsolete' := 'No longer any reason to use this, all state classes can have unit tests.'}
FUNCTION_BLOCK FB_PositionStateInOut_WithPMPS_Test EXTENDS FB_PositionStateBase_WithPMPS_Test
(*
    Example usage of FB_PositionStateBase_WithPMPS_Test for a simple IN/OUT axis. See NOTE: comments.
    Also usable as a drop-in for these cases (no need to roll your own in/out)

    This is the PMPS version. Note that the only difference is that we extend the _WithPMPS_Test FB.
*)
VAR_INPUT
    // The enum position to move to
    {attribute 'pytmc' := '
        pv: SET
        io: io
    '}
    enumSet: ENUM_EpicsInOut_INT; // NOTE: Please copy this pragma exactly on your enumSet

    // Information about the OUT position
    stOut: ST_PositionState; // NOTE: Do not pragma these, let it happen in the manager.
    // Information about the IN position
    stIn: ST_PositionState;
END_VAR
VAR_OUTPUT
    // The enum state readback
    {attribute 'pytmc' := '
        pv: GET
        io: i
    '}
    enumGet: ENUM_EpicsInOut_INT; // NOTE: Please copy this pragma exactly on your enumGet
END_VAR
VAR
    bInOutInit: BOOL;
END_VAR

IF NOT bInOutInit THEN
    bInOutInit := TRUE;
    arrStates[1] := stOut;
    arrStates[2] := stIn;
    stOut.sName := 'OUT';
    stIn.sName := 'IN';
END_IF
setState := enumSet;
Exec();
enumGet := getState;
enumSet := setState;

END_FUNCTION_BLOCK

// POUs/Deprecated/FB_PositionStatePMPS_Test
{attribute 'obsolete' := 'No longer any reason to use this, all state classes can have unit tests.'}
FUNCTION_BLOCK FB_PositionStatePMPS_Test EXTENDS FB_PositionStatePMPS_Base
(*
    Implement position state pmps with no FFO and auto-accept transition after 3s
    Use for offline testing of everything except the explicit interface
*)
VAR
    tonReq: TON;
END_VAR

Exec();

ACTION HandleBPTM:
// Send the fake BPTM our assertion request by changing stStateReq.stBeamParams
// We expect to recieve bTransitionAuthorized TRUE after some delta T
// We expect bTransitionAuthorized to go FALSE after stMotionStage.bBusy goes FALSE
tonReq(
    IN:=bInTransition,
    PT:=T#3s);
bTransitionAuthorized := tonReq.Q AND stMotionStage.bExecute;
END_ACTION

ACTION HandleFFO:
// Skip implementing this for offline testing
// We won't be able to tell if it worked anyway
END_ACTION

END_FUNCTION_BLOCK

// POUs/Deprecated/FB_StatePTPMove
{attribute 'obsolete' := 'Use FB_PositionStateMove instead'}
FUNCTION_BLOCK FB_StatePTPMove
// Do not use, this is deprecated
VAR_INPUT
    {attribute 'pytmc' := '
        pv:
    '}
    stPositionState: ST_PositionState;

    {attribute 'pytmc' := '
        pv: GO
        io: io
        field: ZNAM False
        field: ONAM True
    '}
    bExecute: BOOL;

    bMoveOk: BOOL;
END_VAR
VAR_IN_OUT
    stMotionStage: ST_MotionStage;
END_VAR
VAR_OUTPUT
    {attribute 'pytmc' := '
        pv: AT_STATE
        io: input
        field: ZNAM False
        field: ONAM True
    '}
    bAtState: BOOL;

    {attribute 'pytmc' := '
        pv: DMOV
        io: input
        field: ZNAM False
        field: ONAM True
    '}
    bDone: BOOL;

    {attribute 'pytmc' := '
        pv: BUSY
        io: input
        field: ZNAM False
        field: ONAM True
    '}
    bBusy: BOOL;

    {attribute 'pytmc' := '
        pv: ERR
        io: input
        field: ZNAM False
        field: ONAM True
    '}
    bError: BOOL;

    {attribute 'pytmc' := '
        pv: ERRMSG
        io: input
    '}
    sError: STRING;
END_VAR
VAR
    bExecTrig: R_TRIG;
    bExecEnd: F_TRIG;
    fActPosition: LREAL;
    fLowPos: LREAL;
    fHighPos: LREAL;
END_VAR

bExecTrig(CLK:=bExecute);
IF bExecTrig.Q AND bMoveOk THEN
    IF NOT stMotionStage.bBusy AND NOT stMotionStage.bError THEN
        stMotionStage.bExecute := TRUE;
        stMotionStage.nCommand := E_EpicsMotorCmd.MOVE_ABSOLUTE;
        stMotionStage.fPosition := stPositionState.fPosition;
        stMotionStage.fVelocity := stPositionState.fVelocity;
        stMotionStage.fAcceleration := stPositionState.fAccel;
        stMotionStage.fDeceleration := stPositionState.fDecel;
        bDone := FALSE;
        bBusy := TRUE;
    END_IF
END_IF
bError := stMotionStage.bError;
sError := stMotionStage.sErrorMessage;

fActPosition := stMotionStage.stAxisStatus.fActPosition;
fLowPos := stPositionState.fPosition - stPositionState.fDelta;
fHighPos := stPositionState.fPosition + stPositionState.fDelta;
IF (fLowPos < fActPosition) AND (fHighPos > fActPosition) THEN
    bAtState := TRUE;
    IF NOT stMotionStage.bBusy THEN
        bDone := TRUE;
        bBusy := FALSE;
        bExecute := FALSE;
    END_IF
ELSE
    bAtState := FALSE;
END_IF

bExecEnd(CLK:=bExecute);
IF bExecEnd.Q AND bBusy THEN
    stMotionStage.bExecute := FALSE;
END_IF

IF NOT stMotionStage.bExecute OR NOT bExecute THEN
    bDone := TRUE;
    bBusy := FALSE;
    bExecute := FALSE;
END_IF

END_FUNCTION_BLOCK

// POUs/ImplicitChecks/CheckBounds
// Implicitly generated code : DO NOT EDIT
FUNCTION CheckBounds : DINT
VAR_INPUT
    index, lower, upper: DINT;
END_VAR

// Implicitly generated code : Only an Implementation suggestion
{noflow}
IF  index < lower THEN
    CheckBounds := lower;
ELSIF  index > upper THEN
    CheckBounds := upper;
ELSE
    CheckBounds := index;
END_IF
{flow}

END_FUNCTION

// POUs/ImplicitChecks/CheckDivDInt
// Implicitly generated code : DO NOT EDIT
FUNCTION CheckDivDInt : DINT
VAR_INPUT
    divisor:DINT;
END_VAR

// Implicitly generated code : Only an Implementation suggestion
{noflow}
IF divisor = 0 THEN
    CheckDivDInt:=1;
ELSE
    CheckDivDInt:=divisor;
END_IF;
{flow}

END_FUNCTION

// POUs/ImplicitChecks/CheckDivLInt
// Implicitly generated code : DO NOT EDIT
FUNCTION CheckDivLInt : LINT
VAR_INPUT
    divisor:LINT;
END_VAR

// Implicitly generated code : Only an Implementation suggestion
{noflow}
IF divisor = 0 THEN
    CheckDivLInt:=1;
ELSE
    CheckDivLInt:=divisor;
END_IF;
{flow}

END_FUNCTION

// POUs/ImplicitChecks/CheckDivLReal
// Implicitly generated code : DO NOT EDIT
FUNCTION CheckDivLReal : LREAL
VAR_INPUT
    divisor:LREAL;
END_VAR

// Implicitly generated code : Only an Implementation suggestion
{noflow}
IF divisor = 0 THEN
    CheckDivLReal:=1;
ELSE
    CheckDivLReal:=divisor;
END_IF;
{flow}

END_FUNCTION

// POUs/ImplicitChecks/CheckDivReal
// Implicitly generated code : DO NOT EDIT
FUNCTION CheckDivReal : REAL
VAR_INPUT
    divisor:REAL;
END_VAR

// Implicitly generated code : Only an Implementation suggestion
{noflow}
IF divisor = 0 THEN
    CheckDivReal:=1;
ELSE
    CheckDivReal:=divisor;
END_IF;
{flow}

END_FUNCTION

// POUs/Motion/Gantry/FB_GantryAutoCoupling
FUNCTION_BLOCK FB_GantryAutoCoupling
VAR_INPUT
    nGantryTol : LINT;
END_VAR
VAR_OUTPUT
    bGantryAlreadyCoupled : BOOL;
END_VAR
VAR_IN_OUT
    Master : ST_MotionStage;
    MasterEnc : ST_RenishawAbsEnc;
    Slave : ST_MotionStage;
    SlaveEnc : ST_RenishawAbsEnc;
    bExecuteCouple : BOOL;
    bExecuteDecouple : BOOL;
END_VAR
VAR
    gantry_diff_limit : FB_GantryDiffVirtualLimitSwitch;
    couple : MC_GEARIN;
    decouple : MC_GEAROUT;
    bInitComplete : BOOL;
    fbSetEnables : FB_SetEnables;
END_VAR

// Designate Master and SLave Axes
Master.bGantryAxis := TRUE;
Slave.bGantryAxis := TRUE;

Master.nGantryTol := nGantryTol;
Slave.nGantryTol := Master.nGantryTol;

// Activate Gantry Virtual Limit Switch
gantry_diff_limit(Penc:=MasterEnc, SEnc:=SlaveEnc, GantDiffTol:=Master.nGantryTol,
                  PLimFwd=>Master.bGantryForwardEnable, PLimBwd=>Master.bGantryBackwardEnable,
                  SLimFwd=>Slave.bGantryForwardEnable, SLimBwd=>Slave.bGantryBackwardEnable);

// Coupling Status Bit
bGantryAlreadyCoupled := Master.Axis.NcToPlc.CoupleState=1 AND Slave.Axis.NcToPlc.CoupleState=3;

fbSetEnables(stMotionStage:=Master);
fbSetEnables(stMotionStage:=Slave);

IF bGantryAlreadyCoupled THEN
    Master.bGantryForwardEnable := Master.bGantryForwardEnable AND Slave.bAllForwardEnable;
    Slave.bGantryForwardEnable := Master.bAllForwardEnable AND Slave.bGantryForwardEnable;

    Master.bGantryBackwardEnable := Master.bGantryBackwardEnable AND Slave.bAllBackwardEnable;
    Slave.bGantryBackwardEnable := Master.bAllBackwardEnable AND Slave.bGantryBackwardEnable;
END_IF


// Coupling states
// Auto-coupling at init and auto-reset of coupling boolean
bExecuteCouple S= NOT bInitComplete;

bExecuteCouple R= couple.Busy OR bGantryAlreadyCoupled;
couple(Master:=Master.Axis, Slave:=Slave.Axis, Execute:=bExecuteCouple);

bInitComplete S= bGantryAlreadyCoupled;

// Decoupling with auto-reset of coupling boolean
bExecuteDecouple R= decouple.Busy OR NOT bGantryAlreadyCoupled;
decouple(Slave:=Slave.Axis, Execute:=bExecuteDecouple);

END_FUNCTION_BLOCK

// POUs/Motion/Gantry/FB_GantryDiffVirtualLimitSwitch
FUNCTION_BLOCK FB_GantryDiffVirtualLimitSwitch
VAR_INPUT
    PEnc: ST_RenishawAbsEnc; // Primary axis encoder (usually the upstream one)
    SEnc: ST_RenishawAbsEnc; // Secondary axis encoder (couples to the primary)

    GantDiffTol: LINT;        // Gantry differenace tolerance in encoder counts
END_VAR
VAR_OUTPUT
    PLimFwd: BOOL; // Primary axis forward direction enable
    PLimBwd: BOOL; // Primary axis reverse direction enable
    SLimFwd: BOOL; // Secondary axis forward direction enable
    SLimBwd: BOOL; // Secondary axis reverse direction enable
END_VAR
VAR
    GantryDiff: LINT;
END_VAR

(* Gantry Difference Virtual Limit Switch
A. Wallace 2017-2-15

Determines which direction is disabled due to it increasing the gantry difference.
Refer to the ESD for actual conventions.

A positive gantry error refers to a CCW clocked assembly:
eg. for X
X1 upstream, X2 downstream. Primary axis is always upstream.
Gantry difference > 0 when
X2>X1
Therefore
X2 positive direction disabled
X1 negative direction disabled

Call before FB_MotionStage fb calls for the gantry axes.
*)

GantryDiff := ( ULINT_TO_LINT(PEnc.Count) - ULINT_TO_LINT(PEnc.Ref) ) - ( ULINT_TO_LINT(SEnc.Count) - ULINT_TO_LINT(SEnc.Ref) );

IF ABS(GantryDiff) > GantDiffTol THEN
    IF GantryDiff < 0  THEN
        PLimBwd := FALSE;
        SLimFwd := FALSE;
    ELSE
        PLimBwd := TRUE;
        SLimFwd := TRUE;
    END_IF
    IF GantryDiff > 0 THEN
        PLimFwd := FALSE;
        SLimBwd := FALSE;
    ELSE
        PLimFwd := TRUE;
        SLimBwd := TRUE;
    END_IF
ELSE
    //If there is no fault, all directions are enabled
    PLimFwd := TRUE;
    PLimBwd := TRUE;
    SLimFwd := TRUE;
    SLimBwd := TRUE;
END_IF

END_FUNCTION_BLOCK

// POUs/Motion/PMPS/FB_PositionStatePMPS3D
FUNCTION_BLOCK FB_PositionStatePMPS3D
(*
    3-Dimensional position state function block with PMPS.

    This allows the user to move 3 motors among some set of named state positions with PMPS protection.

    To use a states block, you must define enums that match the state options and give them pytmc pragmas.
    See FB_PositionState1D_InOut for a simple example.
    These enums must be passed in as the eEnumSet and eEnumGet VAR_IN_OUT variables.
    The enum values must match the array indices in astPositionState1, astPositionState2, and astPositionState3.

    A move will begin when eEnumSet is set to a positive, nonzero value. eEnumSet will be reset to 0 on every cycle, allowing us
    to accept a new, possibly conflicting, move request on the next cycle to interrupt the first.

    The motors must already be set up for point-to-point motion via FB_MotionStage, etc., for this function block to work properly.

    PMPS handling is done via database lookups by setting sPmpsState on each position state and on
    the transition state input appropriately.
*)
VAR_IN_OUT
    // The 1st motor to move
    stMotionStage1: ST_MotionStage;
    // The 2nd motor to move
    stMotionStage2: ST_MotionStage;
    // The 3rd motor to move
    stMotionStage3: ST_MotionStage;
    // All possible position states for motor 1, including unused/invalid states.
    {attribute 'pytmc' := '
        pv: STATE:M1
        io: io
        expand: :%.2d
    '}
    astPositionState1: ARRAY[1..GeneralConstants.MAX_STATES] OF ST_PositionState;
    // All possible position states for motor 2, including unused/invalid states.
    {attribute 'pytmc' := '
        pv: STATE:M2
        io: io
        expand: :%.2d
    '}
    astPositionState2: ARRAY[1..GeneralConstants.MAX_STATES] OF ST_PositionState;
    // All possible position states for motor 3, including unused/invalid states.
    {attribute 'pytmc' := '
        pv: STATE:M3
        io: io
        expand: :%.2d
    '}
    astPositionState3: ARRAY[1..GeneralConstants.MAX_STATES] OF ST_PositionState;
    // Set this to a nonzero value to request a new move. It will be reset to zero every cycle. This should be hooked up to a user's EPICS enum input.
    eEnumSet: UINT;
    // The current state index, or zero if we are not at a state. This should be hooked up to a user's EPICS enum output.
    eEnumGet: UINT;
    // The fast fault output to fault to.
    fbFFHWO: FB_HardwareFFOutput;
    // The arbiter to request beam conditions from.
    fbArbiter: FB_Arbiter;
END_VAR
VAR_INPUT
    // Set this to TRUE to enable input state moves, or FALSE to disable them.
    bEnableMotion: BOOL;
    // Set this to TRUE to enable beam parameter checks, or FALSE to disable them.
    bEnableBeamParams: BOOL;
    // Set this to TRUE to enable position limit checks, or FALSE to disable them.
    bEnablePositionLimits: BOOL;
    // The name of the device for use in the PMPS DB lookup and diagnostic screens.
    sDeviceName: STRING;
    // The name of the transition state in the PMPS database.
    sTransitionKey: STRING;
    // Normal EPICS inputs, gathered into a single struct
    {attribute 'pytmc' := 'pv: STATE'}
    // PMPS EPICS inputs, gathered into a single struct
    stEpicsToPlc: ST_StateEpicsToPlc;
    {attribute 'pytmc' := 'pv: STATE'}
    stPMPSEpicsToPlc: ST_StatePMPSEpicsToPlc;
    // Set this to TRUE to re-read the loaded database immediately (useful for debug)
    bReadDBNow: BOOL;
END_VAR
VAR_OUTPUT
    // Normal EPICS outputs, gathered into a single struct
    {attribute 'pytmc' := 'pv: STATE'}
    stPlcToEpics: ST_StatePlcToEpics;
    // PMPS EPICS outputs, gathered into a single struct
    {attribute 'pytmc' := 'pv: STATE'}
    stPMPSPlcToEpics: ST_StatePMPSPlcToEpics;
    // The PMPS database lookup associated with the current position state.
    stDbStateParams: ST_DbStateParams;
END_VAR
VAR
    fbCore: FB_PositionStateND_Core;
    fbPMPSCore: FB_PositionStatePMPSND_Core;
    astMotionStageMax: ARRAY[1..MotionConstants.MAX_STATE_MOTORS] OF ST_MotionStage;
    astPositionStateMax: ARRAY[1..MotionConstants.MAX_STATE_MOTORS] OF ARRAY[1..GeneralConstants.MAX_STATES] OF ST_PositionState;
END_VAR


astMotionStageMax[1] := stMotionStage1;
astMotionStageMax[2] := stMotionStage2;
astMotionStageMax[3] := stMotionStage3;
astPositionStateMax[1] := astPositionState1;
astPositionStateMax[2] := astPositionState2;
astPositionStateMax[3] := astPositionState3;

fbCore(
    astMotionStageMax:=astMotionStageMax,
    astPositionStateMax:=astPositionStateMax,
    stEpicsToPlc:=stEpicsToPlc,
    stPlcToEpics:=stPlcToEpics,
    eEnumSet:=eEnumSet,
    eEnumGet:=eEnumGet,
    bEnable:=bEnableMotion,
    nActiveMotorCount:=3,
    nCurrGoal=>,
);
fbPMPSCore(
    astMotionStageMax:=astMotionStageMax,
    astPositionStateMax:=astPositionStateMax,
    stEpicsToPlc:=stEpicsToPlc,
    stPMPSEpicsToPlc:=stPMPSEpicsToPlc,
    stPlcToEpics:=stPlcToEpics,
    stPMPSPlcToEpics:=stPMPSPlcToEpics,
    fbFFHWO:=fbFFHWO,
    fbArbiter:=fbArbiter,
    bEnableBeamParams:=bEnableBeamParams,
    bEnablePositionLimits:=bEnablePositionLimits,
    nActiveMotorCount:=3,
    sDeviceName:=sDeviceName,
    sTransitionKey:=sTransitionKey,
    nCurrGoal:=fbCore.nCurrGoal,
    bReadDBNow:=bReadDBNow,
    stDbStateParams=>stDbStateParams,
);

stMotionStage1 := astMotionStageMax[1];
stMotionStage2 := astMotionStageMax[2];
stMotionStage3 := astMotionStageMax[3];
astPositionState1 := astPositionStateMax[1];
astPositionState2 := astPositionStateMax[2];
astPositionState3 := astPositionStateMax[3];

END_FUNCTION_BLOCK

// POUs/Motion/PMPS/FB_Standard_PMPSDB
FUNCTION_BLOCK FB_Standard_PMPSDB
(*
    This FB should be run on every motion PLC to encapsulate the pmps file reader.
    It is pre-instantiated at MOTION_GVL.fbStandardPMPSDB
*)
VAR_IN_OUT
    // The fast fault output to fault to.
    io_fbFFHWO: FB_HardwareFFOutput;
END_VAR
VAR_INPUT
    // If TRUE, FB will run. Reads when enable goes TRUE.
    bEnable: BOOL;
    // E.g. lfe-motion
    sPlcName: STRING;
    {attribute 'pytmc' := '
        pv: REFRESH
        io: io
    '}
    // Set to TRUE to cause an extra read.
    bRefresh: BOOL;
    // Directory where the DB is stored.
    sDirectory: STRING := '';
END_VAR
VAR_OUTPUT
    {attribute 'pytmc' := '
        pv: LAST_REFRESH
        io: i
    '}
    nLastRefreshTime: DINT;
    bReadPmpsDb: BOOL;
END_VAR
VAR
    bExecute: BOOL;
    rtEnable: R_TRIG;
    rtRefresh: R_TRIG;
    ftBusy: F_TRIG;

    // Time tracking liften from Arbiter PLCs
    fbTime : FB_LocalSystemTime := ( bEnable := TRUE, dwCycle := 1 );
    fbTime_to_UTC: FB_TzSpecificLocalTimeToSystemTime;
    fbGetTimeZone: FB_GetTimeZoneInformation;

    fbIPCReg: FB_IPCDiag_Register;
    fbCheckOS: FB_IPCDiag_ReadParameter;
    sOSName: STRING := '';
    nCheckOSTries: UINT := 3;
END_VAR

IF NOT bEnable THEN
    RETURN;
END_IF

rtEnable(CLK:=bEnable);
rtRefresh(CLK:=bRefresh);
bRefresh := FALSE;

IF rtEnable.Q OR rtRefresh.Q THEN
    // Make sure file reader gets a rising edge
    MOTION_GVL.fbPmpsFileReader(
        io_fbFFHWO:=io_fbFFHWO,
        bExecute:=FALSE,
    );
    bExecute := TRUE;
END_IF

IF sDirectory = '' THEN
    // Check OS for default directory
    fbIPCReg(
        bExecute:=TRUE,
        tTimeout:=T#1s,
    );
    fbCheckOS(
        bExecute:=fbIPCReg.bValid,
        eParameterKey:=E_IPCDiag_ParameterKey.OS_Name,
        fbRegister:=fbIPCReg,
    );
    IF fbIPCReg.bError OR fbCheckOS.bError THEN
        IF nCheckOSTries <= 0 THEN
            // Retry counter down to zero: set to error name to try old default
            sOSName := 'Error';
        ELSE
            // Decrement retry counter
            nCheckOSTries := nCheckOSTries - 1;
            // Reset FBs
            fbCheckOS(bExecute:=FALSE, fbRegister:=fbIPCReg);
            fbIPCReg(bExecute:=FALSE);
        END_IF
    ELSIF fbCheckOS.bValid THEN
        fbCheckOS.GetParameter(
            pBuffer:=ADR(sOSName),
            nBufferSize:=SIZEOF(sOSName),
        );
    END_IF
    IF sOSName = 'TwinCAT/BSD' THEN
        sDirectory := '/home/ecs-user/pmpsdb/';
    ELSIF sOSName <> '' THEN
        sDirectory := '/Hard Disk/ftp/PMPS/';
    END_IF
END_IF

MOTION_GVL.fbPmpsFileReader(
    io_fbFFHWO:=io_fbFFHWO,
    bExecute:=bExecute AND sDirectory <> '',
    sSrcPathName:=CONCAT(CONCAT(sDirectory, sPlcName), '.json'),
    sPLCName:=sPLCName,
    PMPS_jsonDoc=>PMPS_GVL.BP_jsonDoc,
);

ftBusy(CLK:=MOTION_GVL.fbPmpsFileReader.bBusy);
IF ftBusy.Q THEN
    bReadPmpsDb := TRUE;
ELSE
    bReadPmpsDb := FALSE;
END_IF


// Lifted from Arbiter PLCs: keep track of the time
fbTime(sNetID:='');
fbGetTimeZone(sNetID:='', bExecute:=TRUE, tTimeout:=T#10S);
fbTime_to_UTC(in:= fbTime.systemTime , tzInfo:=fbGetTimeZone.tzInfo);

// Update the refresh time on successful read
IF ftBusy.Q AND NOT MOTION_GVL.fbPmpsFileReader.bError THEN
   nLastRefreshTime := TO_DINT(TO_DT(SystemTime_TO_DT(fbTime_to_UTC.out)));
END_IF

bExecute R= ftBusy.Q;

END_FUNCTION_BLOCK

// POUs/Motion/States/Examples/FB_PositionState2D_InOut
FUNCTION_BLOCK FB_PositionState2D_InOut
(*
    An example and usable drop-in instance for a 2D state device with just an IN and an OUT state.
*)
VAR_IN_OUT
    // Include stages that can be passed into the FB
    stMotionStage1: ST_MotionStage;
    stMotionStage2: ST_MotionStage;
    // Simplify the interface, the user just needs to construct and pass in and out position states
    stIn1: ST_PositionState;
    stOut1: ST_PositionState;
    stIn2: ST_PositionState;
    stOut2: ST_PositionState;
END_VAR
VAR_INPUT
    // Define an ENUM for EPICS to use to set a new value. It is expected this will be written to during one cycle, so don't continually apply a value here in the PLC code.
    // It is exposed as an input so we can test it using the PLC.
    {attribute 'pytmc' := '
      pv: STATE:SET
      io: io
    '}
    eStateSet: E_EpicsInOut;
END_VAR
VAR_OUTPUT
    // Define an ENUM for EPICS to use to report the new value.
    {attribute 'pytmc' := '
      pv: STATE:GET
      io: i
    '}
    eStateGet: E_EpicsInOut;
END_VAR
VAR
    // Include the standard fb with blank pv pragma
    {attribute 'pytmc' := 'pv:'}
    fbPositionState2D: FB_PositionState2D;
    // The standard fb expects a full array of position states per motor
    astPositionState1: ARRAY[1..GeneralConstants.MAX_STATES] OF ST_PositionState;
    astPositionState2: ARRAY[1..GeneralConstants.MAX_STATES] OF ST_PositionState;
END_VAR


// Optional: default state names
IF stIn1.sName = '' THEN
    stIn1.sName := 'IN';
END_IF
IF stOut1.sName = '' THEN
    stOut1.sName := 'OUT';
END_IF
IF stIn2.sName = '' THEN
    stIn2.sName := 'IN';
END_IF
IF stOut2.sName = '' THEN
    stOut2.sName := 'OUT';
END_IF

// Assemble the states arrays, matching the enum values
astPositionState1[E_EpicsInOut.OUT] := stOut1;
astPositionState1[E_EpicsInOut.IN] := stIn1;
astPositionState2[E_EpicsInOut.OUT] := stOut2;
astPositionState2[E_EpicsInOut.IN] := stIn2;

// Call the main function block, passing our motors, states, and an enable
fbPositionState2D(
    stMotionStage1:=stMotionStage1,
    astPositionState1:=astPositionState1,
    stMotionStage2:=stMotionStage2,
    astPositionState2:=astPositionState2,
    eEnumSet:=eStateSet,
    eEnumGet:=eStateGet,
    bEnable:=TRUE,
);

// Send updates made on the array back to the inputs (VAR_IN_OUT) for maximum clarity
stOut1 := astPositionState1[E_EpicsInOut.OUT];
stIn1 := astPositionState1[E_EpicsInOut.IN];
stOut2 := astPositionState2[E_EpicsInOut.OUT];
stIn2 := astPositionState2[E_EpicsInOut.IN];

END_FUNCTION_BLOCK

// POUs/Motion/States/Examples/FB_PositionStatePMPS2D_InOut
FUNCTION_BLOCK FB_PositionStatePMPS2D_InOut
(*
    An example and usable drop-in instance for a 2D state device with just an IN and an OUT state.
    Note that the outward-facing API is nearly identical to the non-PMPS version
*)
VAR_IN_OUT
    // Include stages that can be passed into the FB
    stMotionStage1: ST_MotionStage;
    stMotionStage2: ST_MotionStage;
    // Simplify the interface, the user just needs to construct and pass in and out position states
    stIn1: ST_PositionState;
    stOut1: ST_PositionState;
    stIn2: ST_PositionState;
    stOut2: ST_PositionState;
    // Include PMPS output helpers
    fbFFHWO: FB_HardwareFFOutput;
    fbArbiter: FB_Arbiter;
END_VAR
VAR_INPUT
    // Define an ENUM for EPICS to use to set a new value. It is expected this will be written to during one cycle, so don't continually apply a value here in the PLC code.
    // It is exposed as an input so we can test it using the PLC.
    {attribute 'pytmc' := '
      pv: STATE:SET
      io: io
    '}
    eStateSet: E_EpicsInOut;
END_VAR
VAR_OUTPUT
    // Define an ENUM for EPICS to use to report the new value.
    {attribute 'pytmc' := '
      pv: STATE:GET
      io: i
    '}
    eStateGet: E_EpicsInOut;
END_VAR
VAR
    // Include the standard fb with blank pv pragma
    {attribute 'pytmc' := 'pv:'}
    fbPositionStatePMPS2D: FB_PositionStatePMPS2D;
    // The standard fb expects a full array of position states per motor
    astPositionState1: ARRAY[1..GeneralConstants.MAX_STATES] OF ST_PositionState;
    astPositionState2: ARRAY[1..GeneralConstants.MAX_STATES] OF ST_PositionState;
END_VAR


// Optional: default state names
IF stIn1.sName = '' THEN
    stIn1.sName := 'IN';
END_IF
IF stOut1.sName = '' THEN
    stOut1.sName := 'OUT';
END_IF
IF stIn2.sName = '' THEN
    stIn2.sName := 'IN';
END_IF
IF stOut2.sName = '' THEN
    stOut2.sName := 'OUT';
END_IF

// Assemble the states arrays, matching the enum values
astPositionState1[E_EpicsInOut.OUT] := stOut1;
astPositionState1[E_EpicsInOut.IN] := stIn1;
astPositionState2[E_EpicsInOut.OUT] := stOut2;
astPositionState2[E_EpicsInOut.IN] := stIn2;

// Call the main function block, passing our motors, states, and an enable
fbPositionStatePMPS2D(
    fbFFHWO:=fbFFHWO,
    fbArbiter:=fbArbiter,
    stMotionStage1:=stMotionStage1,
    astPositionState1:=astPositionState1,
    stMotionStage2:=stMotionStage2,
    astPositionState2:=astPositionState2,
    eEnumSet:=eStateSet,
    eEnumGet:=eStateGet,
    bEnableMotion:=TRUE,
    bEnableBeamParams:=TRUE,
    bEnablePositionLimits:=TRUE,
);

// Send updates made on the array back to the inputs (VAR_IN_OUT) for maximum clarity
stOut1 := astPositionState1[E_EpicsInOut.OUT];
stIn1 := astPositionState1[E_EpicsInOut.IN];
stOut2 := astPositionState2[E_EpicsInOut.OUT];
stIn2 := astPositionState2[E_EpicsInOut.IN];

END_FUNCTION_BLOCK

// POUs/Motion/States/FB_PositionState3D
FUNCTION_BLOCK FB_PositionState3D
(*
    3-Dimensional position state function block.

    This allows the user to move 3 motors among some set of named state positions.

    To use a states block, you must define enums that match the state options and give them pytmc pragmas.
    See FB_PositionState1D_InOut for a simple example.
    These enums must be passed in as the eEnumSet and eEnumGet VAR_IN_OUT variables.
    The enum values must match the array indices in astPositionState1, astPositionState2, and astPositionState3.

    A move will begin when eEnumSet is set to a positive, nonzero value. eEnumSet will be reset to 0 on every cycle, allowing us
    to accept a new, possibly conflicting, move request on the next cycle to interrupt the first.

    The motors must already be set up for point-to-point motion via FB_MotionStage, etc., for this function block to work properly.

    With no PMPS handling, this FB basically just links the state names with positions in both directions for set and readback.
*)
VAR_IN_OUT
    // The 1st motor to move
    stMotionStage1: ST_MotionStage;
    // The 2nd motor to move
    stMotionStage2: ST_MotionStage;
    // The 3rd motor to move
    stMotionStage3: ST_MotionStage;
    // All possible position states for motor 1, including unused/invalid states.
    {attribute 'pytmc' := '
        pv: STATE:01
        io: io
        expand: :%.2d
    '}
    astPositionState1: ARRAY[1..GeneralConstants.MAX_STATES] OF ST_PositionState;
    // All possible position states for motor 2, including unused/invalid states.
    {attribute 'pytmc' := '
        pv: STATE:02
        io: io
        expand: :%.2d
    '}
    astPositionState2: ARRAY[1..GeneralConstants.MAX_STATES] OF ST_PositionState;
    // All possible position states for motor 3, including unused/invalid states.
    {attribute 'pytmc' := '
        pv: STATE:03
        io: io
        expand: :%.2d
    '}
    astPositionState3: ARRAY[1..GeneralConstants.MAX_STATES] OF ST_PositionState;
    // Set this to a nonzero value to request a new move. It will be reset to zero every cycle. This should be hooked up to a user's EPICS enum input.
    eEnumSet: UINT;
    // The current state index, or zero if we are not at a state. This should be hooked up to a user's EPICS enum output.
    eEnumGet: UINT;
END_VAR
VAR_INPUT
    // Set this to TRUE to enable input state moves, or FALSE to disable them.
    bEnable: BOOL;
    // Normal EPICS inputs, gathered into a single struct
    {attribute 'pytmc' := 'pv: STATE'}
    stEpicsToPlc: ST_StateEpicsToPlc;
END_VAR
VAR_OUTPUT
    // Normal EPICS outputs, gathered into a single struct
    {attribute 'pytmc' := 'pv: STATE'}
    stPlcToEpics: ST_StatePlcToEpics;
END_VAR
VAR
    fbCore: FB_PositionStateND_Core;
    astMotionStageMax: ARRAY[1..MotionConstants.MAX_STATE_MOTORS] OF ST_MotionStage;
    astPositionStateMax: ARRAY[1..MotionConstants.MAX_STATE_MOTORS] OF ARRAY[1..GeneralConstants.MAX_STATES] OF ST_PositionState;
END_VAR


astMotionStageMax[1] := stMotionStage1;
astMotionStageMax[2] := stMotionStage2;
astMotionStageMax[3] := stMotionStage3;
astPositionStateMax[1] := astPositionState1;
astPositionStateMax[2] := astPositionState2;
astPositionStateMax[3] := astPositionState3;

fbCore(
    astMotionStageMax:=astMotionStageMax,
    astPositionStateMax:=astPositionStateMax,
    stEpicsToPlc:=stEpicsToPlc,
    stPlcToEpics:=stPlcToEpics,
    eEnumSet:=eEnumSet,
    eEnumGet:=eEnumGet,
    bEnable:=bEnable,
    nActiveMotorCount:=3,
);

stMotionStage1 := astMotionStageMax[1];
stMotionStage2 := astMotionStageMax[2];
stMotionStage3 := astMotionStageMax[3];
astPositionState1 := astPositionStateMax[1];
astPositionState2 := astPositionStateMax[2];
astPositionState3 := astPositionStateMax[3];

END_FUNCTION_BLOCK

// POUs/Motion/States/FB_StateSetupHelper
FUNCTION_BLOCK FB_StateSetupHelper
(*
    This is a helper for setting up large numbers of ST_PositionState instances.

    This is typically verbose to do by hand in the normal ways and can be error-prone.

    Calling with bSetDefault:=TRUE will set the default values to all the values
    from the input stPositionState. Note that the other args will be ignored in this case.
    This must be done at least once. If you forget to do this, there will be a warning and
    bValid will be set to FALSE, making it so we cannot move to that state.

    Calling without bSetDefault or with it set to FALSE will apply values to the
    input stPositionState with the following priority order:

    1. The value used in the function block call
    2. The value from the template stPositionState used in the most recent
       call with bSetDefault:=TRUE
    3. The original default value as defined on ST_PositionState

    For ease of use, to enable EPICS writes if unlocked, and to avoid repeated
    self-overwrites in the encoder count use case, this function block will not
    reapply the values to the same state again after the state has been fully
    initialized by the states function blocks, as determined by the bUpdated struct
    member. If you want to force the function block to reapply every cycle you can
    set bForceUpdate to TRUE, but it is not recommended. Without this feature,
    you would be required to wrap this function block in a guard to make sure it
    was only called once per state, which is fairly annoying.

    Example expected usage:
    VAR
        fbStateSetup: FB_StateSetupHelper;
        stDefault: ST_PositionState := (
            fDelta := 0.5,
            fVelocity := 10,
            bMoveOk := TRUE,
            bValid := TRUE
        );
        astStates1: ARRAY[1..GeneralConstants.MAX_STATES] OF ST_PositionState;
        astStates2: ARRAY[1..GeneralConstants.MAX_STATES] OF ST_PositionState;
        astStates2: ARRAY[1..GeneralConstants.MAX_STATES] OF ST_PositionState;
    END_VAR

    fbStateSetup(stPositionState:=stDefault, bSetDefault:=TRUE);

    fbStateSetup(stPositionState:=astStates1[1], sName:='OUT', fPosition:=10);
    fbStateSetup(stPositionState:=astStates1[2], sName:='YAG', fPosition:=20);
    fbStateSetup(stPositionState:=astStates1[3], sName:='TT', fPosition:=30);

    fbStateSetup(stPositionState:=astStates2[1], sName:='OUT', fPosition:=-30);
    fbStateSetup(stPositionState:=astStates2[2], sName:='YAG', fPosition:=35);
    fbStateSetup(stPositionState:=astStates2[3], sName:='TT', fPosition:=70);

    fbStateSetup(stPositionState:=astStates3[1], sName:='OUT', fPosition:=0.4, fDelta:=0.1);
    fbStateSetup(stPositionState:=astStates3[2], sName:='YAG', fPosition:=2.3, fDelta:=0.1);
    fbStateSetup(stPositionState:=astStates3[3], sName:='TT', fPosition:=5.6, fDelta:=0.1;
*)
VAR_IN_OUT
    stPositionState: ST_PositionState;
END_VAR
VAR_INPUT
    bSetDefault: BOOL;
    bForceUpdate: BOOL;
    sName: STRING;
    fPosition: LREAL;
    nEncoderCount: UDINT;
    fDelta: LREAL;
    fVelocity: LREAL;
    fAccel: LREAL;
    fDecel: LREAL;
    bMoveOk: BOOL;
    bLocked: BOOL;
    bValid: BOOL;
    bUseRawCounts: BOOL;
    sPmpsState: STRING;
END_VAR
VAR
    stDefault: ST_PositionState;
    fbWarning: FB_LogMessage;
    bHasDefault: BOOL;
    bHasWarned: BOOL;
    sJson: STRING;
END_VAR


IF bSetDefault THEN
    bSetDefault := FALSE;
    bHasDefault := TRUE;
    stDefault := stPositionState;
ELSIF bForceUpdate OR NOT stPositionState.bUpdated THEN
    stPositionState.sName := sName;
    stPositionState.fPosition := fPosition;
    stPositionState.nEncoderCount := nEncoderCount;
    stPositionState.fDelta := fDelta;
    stPositionState.fVelocity := fVelocity;
    stPositionState.fAccel := fAccel;
    stPositionState.fDecel := fDecel;
    stPositionState.bMoveOk := bMoveOk;
    stPositionState.bLocked := bLocked;
    stPositionState.bValid := bValid;
    stPositionState.bUseRawCounts := bUseRawCounts;
    stPositionState.stPMPS.sPmpsState := sPmpsState;
    IF NOT bHasDefault THEN
        stPositionState.bValid := FALSE;
        IF NOT bHasWarned THEN
            bHasWarned := TRUE;
            sJson := CONCAT(CONCAT(CONCAT(CONCAT('{"sName": "', sName), '", "sPmpsState": "'), sPmpsState), '"}');
            fbWarning(
                sMsg:=CONCAT('Did not initialize any defaults in FB_StateSetupHelper! Some states are disabled, check your code! ', sJson),
                eSevr:=TcEventSeverity.Warning,
                eSubSystem:=E_Subsystem.MOTION,
                sJson:=sJson,
            );
        END_IF
    END_IF
END_IF

// Overwrite the input args so that unset args are the defaults in the next call
sName := stDefault.sName;
fPosition := stDefault.fPosition;
nEncoderCount := stDefault.nEncoderCount;
fDelta := stDefault.fDelta;
fVelocity := stDefault.fVelocity;
fAccel := stDefault.fAccel;
fDecel := stDefault.fDecel;
bMoveOk := stDefault.bMoveOk;
bLocked := stDefault.bLocked;
bValid := stDefault.bValid;
bUseRawCounts := stDefault.bUseRawCounts;
sPmpsState := stDefault.stPMPS.sPmpsState;

END_FUNCTION_BLOCK

// POUs/Motion/FB_MotionPneumaticActuator
(*This function blcok implements a pnuematic actuator. That can be signle or double acting by setting the ibSingleCntrl accordingly*)
(* with double acting ibCntrlHold signal should be false, while with single acting the signal should be true*)
FUNCTION_BLOCK FB_MotionPneumaticActuator
VAR_INPUT
    (*EPS Interlock Bits*)
    ibInsertOK: BOOL; (*Actuator can be Inserted*)
    ibRetractOK: BOOL; (*ACtuator can be retracted*)
    ibPMPS_OK:BOOL; (*to be linked the Arbiter bit*)
    ibSingleCntrl:BOOL;(* TRUE if Actuator requires one Output signal to be activated, FALSE if its double acting i.e two outputs are required*)
    ibCntrlHold:BOOL; (* Control Signal must retain its value, must be TRUE in the case of single acting*)
    ibOverrideInterlock:BOOL; (*if true interlocks are ignored*)
    // Reset fault
    {attribute 'pytmc' := '
    pv: FFO_Reset
    '}
    i_xReset: BOOL;
    {attribute 'pytmc' := '
    pv: FFO_AutoReset
    '}
    i_xAutoReset: BOOL;
END_VAR
VAR_OUTPUT
    {attribute 'pytmc' := '
    pv:
    '}
    stPneumaticActuator    :    ST_MotionPneumaticActuator;
    {attribute 'pytmc' := '
     pv: MPS_OK
     field: ZNAM FALSE
     field: ONAM TRUE
     field: DESC TRUE if MPS signal is OK
    '}
    xMPS_OK:BOOL;
END_VAR
VAR_IN_OUT
    io_fbFFHWO    :    FB_HardwareFFOutput;
END_VAR
VAR
    // PMPS
    fbFF    :    FB_FastFault :=(
        i_DevName := 'MPA',
        i_Desc := 'Fault occurs when the device is moving',
        i_TypeCode := E_MotionFFType.PNEUMATIC_MOVE);

    (*Init*)
    xFirstPass    :    BOOL;
    fbFSInit        :    R_TRIG;

    (* Timeouts*)
    tTimeOutDuration: TIME:= T#10S;
    tInserttimeout: TON;
    tRetracttimeout:TON;
    (*Limit switch latch timer*)
    tLimitSwitchLatchDuration: TIME:=T#1S;
    tInsertLimitSwitch:TON;
    tRetractLimitSwitch:TON;

    (*Logging*)
    fbLogger : FB_LogMessage := (eSubsystem:=E_SubSystem.MOTION);
    ePrevState : E_PnuematicActuatorPositionState;
    tAction : R_TRIG; // Primary action of this device (Insert_DO, Retract_DO, etc.)
    tOverrideActivated : R_TRIG;

    (*IO*)
    i_xInsertedLS    AT%I*: BOOL;
    i_xRetractedLS    AT%I*: BOOL;
    q_xInsert_DO    AT%Q*: BOOL;
    q_xRetract_DO    AT%Q*: BOOL;

END_VAR


(*Initialize*)
fbFSInit( CLK := TRUE, Q => xFirstPass);
IF xFirstPass THEN
    stPneumaticActuator.eState := E_PnuematicActuatorPositionState.INVALID;
    stPneumaticActuator.bRetract_SW := FALSE;
    stPneumaticActuator.bInsert_SW := FALSE;
END_IF

(*Soft IO Mapping to EPICS PVs*)
ACT_IO();

(* Manage States*)
IF stPneumaticActuator.i_bInLimitSwitch AND  stPneumaticActuator.i_bOutLimitSwitch THEN
    stPneumaticActuator.eState:=E_PnuematicActuatorPositionState.INVALID;
ELSIF NOT stPneumaticActuator.i_bInLimitSwitch AND stPneumaticActuator.i_bOutLimitSwitch THEN
    stPneumaticActuator.eState:=E_PnuematicActuatorPositionState.RETRACTED;
ELSIF stPneumaticActuator.i_bInLimitSwitch AND NOT stPneumaticActuator.i_bOutLimitSwitch THEN
    stPneumaticActuator.eState:=E_PnuematicActuatorPositionState.INSERTED;
ELSIF NOT stPneumaticActuator.i_bInLimitSwitch AND NOT stPneumaticActuator.i_bOutLimitSwitch THEN
    stPneumaticActuator.eState:=E_PnuematicActuatorPositionState.MOVING;
ELSE
    stPneumaticActuator.eState:=E_PnuematicActuatorPositionState.INVALID ;
END_IF

(*Set the Done/Busy signal*)
stPneumaticActuator.bDone := (stPneumaticActuator.bRetract_SW AND stPneumaticActuator.eState=E_PnuematicActuatorPositionState.RETRACTED)
                            OR (stPneumaticActuator.bInsert_SW AND stPneumaticActuator.eState=E_PnuematicActuatorPositionState.INSERTED);
stPneumaticActuator.bBusy := (stPneumaticActuator.bRetract_SW AND stPneumaticActuator.eState<>E_PnuematicActuatorPositionState.RETRACTED)
                            OR (stPneumaticActuator.bInsert_SW AND stPneumaticActuator.eState<>E_PnuematicActuatorPositionState.INSERTED);
(*MPS FAULT*)
(* MPS Faults when the actuator is in motion*)
xMPS_OK := (stPneumaticActuator.eState=E_PnuematicActuatorPositionState.RETRACTED) OR (stPneumaticActuator.eState=E_PnuematicActuatorPositionState.INSERTED);
(*PMPS PERMISSION*)
// yet to be implemented

(* Can't have bRetract_SW and  bInsert_SW both be true*)
If (stPneumaticActuator.bRetract_SW) AND (stPneumaticActuator.bInsert_SW) THEN
    stPneumaticActuator.bRetract_SW := FALSE;
    stPneumaticActuator.bInsert_SW := FALSE;
END_IF
//Redundant??
(*Check if both digital outputs active at the same time, and clear all*)
IF stPneumaticActuator.q_bInsert THEN
    stPneumaticActuator.q_bRetract := FALSE;
    stPneumaticActuator.bRetract_SW:= FALSE;
END_IF;
IF stPneumaticActuator.q_bRetract THEN
    stPneumaticActuator.q_bInsert := FALSE;
    stPneumaticActuator.bInsert_SW:= FALSE;
END_IF;

(*Actuate the device*)
stPneumaticActuator.q_bRetract := stPneumaticActuator.bRetractOK AND stPneumaticActuator.bRetract_SW AND NOT stPneumaticActuator.bInsert_SW ;
stPneumaticActuator.q_bInsert := stPneumaticActuator.bInsertOK AND stPneumaticActuator.bInsert_SW AND NOT stPneumaticActuator.bRetract_SW ;

(*Reset the Control signal when command has been executed and give time to ensure the actuator is fully seated in either direction*)
IF (NOT ibSingleCntrl AND NOT ibCntrlHold) THEN
   IF (stPneumaticActuator.bRetract_SW AND stPneumaticActuator.i_bOutLimitSwitch AND tRetractLimitSwitch.Q ) THEN stPneumaticActuator.q_bRetract := FALSE; END_IF
   IF (stPneumaticActuator.bInsert_SW AND stPneumaticActuator.i_bInLimitSwitch AND tInsertLimitSwitch.Q) THEN stPneumaticActuator.q_bInsert := FALSE; END_IF
END_IF

(*Timers*)
tInserttimeout(IN:= stPneumaticActuator.q_bInsert, PT := tTimeOutDuration );
tRetracttimeout(IN:= stPneumaticActuator.q_bRetract, PT := tTimeOutDuration);
tInsertLimitSwitch(IN:= stPneumaticActuator.i_bInLimitSwitch, PT := tLimitSwitchLatchDuration);
tRetractLimitSwitch(IN:= stPneumaticActuator.i_bOutLimitSwitch, PT := tLimitSwitchLatchDuration);


///Check moving postion timout
IF NOT stPneumaticActuator.i_bInLimitSwitch AND tInserttimeout.Q THEN
    stPneumaticActuator.bError := TRUE;
    stPneumaticActuator.sErrorMessage:= 'Actuator insert timeout';
ELSIF NOT stPneumaticActuator.i_bOutLimitSwitch AND tRetracttimeout.Q THEN
    stPneumaticActuator.bError := TRUE;
    stPneumaticActuator.sErrorMessage:= 'Actuator retract timeout';
END_IF
// Reset error
stPneumaticActuator.bError R= stPneumaticActuator.bReset;

(*FAST FAULT*)
fbFF(i_xOK := xMPS_OK,
    i_xReset := i_xReset,
    i_xAutoReset := i_xAutoReset,
    io_fbFFHWO := io_fbFFHWO);

(*Soft IO Mapping to Epics pvs*)
ACT_IO();

ACTION ACT_IO:
(*Inputs*)
stPneumaticActuator.i_bInLimitSwitch :=  i_xInsertedLS;
stPneumaticActuator.i_bOutLimitSwitch := i_xRetractedLS;

(*outputs*)
q_xInsert_DO:=stPneumaticActuator.q_bInsert;
q_xRetract_DO:=stPneumaticActuator.q_bRetract;

(*EPICS*)
stPneumaticActuator.bRetractOK := ibRetractOK;
stPneumaticActuator.bInsertOK := ibInsertOK;
END_ACTION

ACTION ACT_Logger:
// Log Valve timeouts
IF (tInserttimeout.Q OR tRetracttimeout.Q) THEN fbLogger(sMsg:=stPneumaticActuator.sErrorMessage, eSevr:=TcEventSeverity.Warning); END_IF

// Log Actuator commands
// Log valve open
tAction(CLK:= (stPneumaticActuator.q_bRetract OR stPneumaticActuator.q_bInsert));
IF tAction.Q THEN
   IF(stPneumaticActuator.q_bRetract) THEN fbLogger(sMsg:='Actuator commanded retract', eSevr:=TcEventSeverity.Info); END_IF
   IF(stPneumaticActuator.q_bInsert) THEN fbLogger(sMsg:='Actuator commanded insert', eSevr:=TcEventSeverity.Info); END_IF
END_IF


// State Logging
IF ePrevState <> stPneumaticActuator.eState THEN
      CASE stPneumaticActuator.eState OF
        E_PnuematicActuatorPositionState.INVALID:
            fbLogger(sMsg:='Actuator invalid position.', eSevr:=TcEventSeverity.Critical);
          E_PnuematicActuatorPositionState.MOVING:
            fbLogger(sMsg:='Actuator moving', eSevr:=TcEventSeverity.Warning);
        E_PnuematicActuatorPositionState.RETRACTED:
            fbLogger(sMsg:='Actuator Retracted.', eSevr:=TcEventSeverity.Info);
        E_PnuematicActuatorPositionState.INSERTED:
            fbLogger(sMsg:='Actuator Inserted.', eSevr:=TcEventSeverity.Info);
      END_CASE
      ePrevState := stPneumaticActuator.eState;
  END_IF
END_ACTION

END_FUNCTION_BLOCK

// POUs/Motion/FB_MotionStageSim
FUNCTION_BLOCK FB_MotionStageSim
(*
    Set all the values needed for a fake motor to be movable
    via the IOC, then call FB_MotionStage
*)
VAR_IN_OUT
    stMotionStage: ST_MotionStage;
END_VAR
VAR_INPUT
    nEnableMode: E_StageEnableMode := E_StageEnableMode.ALWAYS;
END_VAR
VAR
    fbMotionStage: FB_MotionStage;
    bInit: BOOL;
END_VAR

IF NOT bInit THEN
    bInit := TRUE;
    // Stand-in for no forward limit
    stMotionStage.bLimitForwardEnable := TRUE;
    // Stand-in for no reverse limit
    stMotionStage.bLimitBackwardEnable := TRUE;
    // Stand-in for no STO button
    stMotionStage.bHardwareEnable := TRUE;
    // Stand-in for no PMPS governer
    stMotionStage.bPowerSelf := TRUE;
    // Always keep it enabled for testing ease
    stMotionStage.nEnableMode := nEnableMode;
END_IF
// Call FB_MotionStage to do the thing
fbMotionStage(stMotionStage := stMotionStage);

END_FUNCTION_BLOCK

// POUs/Motion/FB_MotionVirtualFrame

FUNCTION_BLOCK FB_MotionVirtualFrame
(*
Takes 3 ST_MotionStages representing real axes that are orthogonal to each other and in a base frame of reference.
Takes 3 ST_MotionStages representing virtual axes that are orthogonal to each other and in a new frame of reference.
Computes the transformation from the base to the new frame of reference using 3 euler angles and a rotation order
as inputs. By default, the order and angles are interpreted as going from the base to the virtual frame. Can be
switched to go from virtual to base frame of reference.
If enabled, this function block will automatically handle commanding the real axes to move when the virtual axes
are commanded to move. If not enabled, the function block acts as a calculator, outputing the results of
calculating motions in a new frame of reference, but not changing any setpoints or commanding any moves.
*)
VAR_IN_OUT
    stMotionStageRx : ST_MotionStage; // Real X Axis in base frame of reference
    stMotionStageRy : ST_MotionStage; // Real Y Axis in base frame of reference
    stMotionStageRz : ST_MotionStage; // Real Z Axis in base frame of reference
    stMotionStageVx : ST_MotionStage; // Virtual X Axis in new frame of reference
    stMotionStageVy : ST_MotionStage; // Virtual Y Axis in new frame of reference
    stMotionStageVz : ST_MotionStage; // Virtual Z Axis in new frame of reference
END_VAR
VAR_INPUT
    (*TRUE to automatically overwrite real axis setpoints and command moves.
      FALSE to use this function only as a calculator.*)
    bEnable : BOOL;
    fAlphaDegrees : LREAL; // Angle of rotation about first axis.
    fBetaDegrees : LREAL; // Angle of rotation about second axis.
    fGammaDegrees : LREAL; // Angle of rotation about third axis.
    (*Rotation Order. E.g: XYZ to rotate alpha degrees around X axis, beta degrees around Y axis,
      and gamma degrees around Z axis. Valid rotation orders are:
      YZY, YXY, ZYZ, ZXZ, XYX, XZX, XYZ, YZX, ZXY, XZY, ZYX, YXZ.
      Default order for empty or invalid input is: ZYX.*)
    sOrder : STRING;
    (*FALSE to define inputs as rotating the frame of reference from the new frame to the base frame.
      TRUE to define the inputs as rotating the frame of reference from the base from to the new frame.*)
    bBaseToNew : BOOL := TRUE;
END_VAR
VAR_OUTPUT
    fbVirtActPositionVec3 : FB_Vec3;
    fbVirtActVelocityVec3 : FB_Vec3;
    fbVirtActAcceleraVec3 : FB_Vec3;

    fbRealTarPositionVec3 : FB_Vec3;
    fbRealTarVelocityVec3 : FB_Vec3;
    fbRealTarAcceleraVec3 : FB_Vec3;
END_VAR
VAR
    fAlphaRadians : LREAL;
    fBetaRadians : LREAL;
    fGammaRadians : LREAL;

    rtExecuteVx : R_TRIG;
    rtExecuteVy : R_TRIG;
    rtExecuteVz : R_TRIG;

    fbRealActPositionVec3 : FB_Vec3;
    fbRealActVelocityVec3 : FB_Vec3;
    fbRealActAcceleraVec3 : FB_Vec3;

    sOrderReversed : STRING;
    sLeft : STRING;
    sMid : STRING;
    sRight : STRING;

    fbVirtTarPositionVec3 : FB_Vec3;
    fbVirtTarVelocityVec3 : FB_Vec3;
    fbVirtTarAcceleraVec3 : FB_Vec3;
END_VAR


fAlphaRadians := DegToRad(fAlphaDegrees);
fBetaRadians := DegToRad(fBetaDegrees);
fGammaRadians := DegToRad(fGammaDegrees);

rtExecuteVx(CLK := stMotionStageVx.bExecute);
rtExecuteVy(CLK := stMotionStageVy.bExecute);
rtExecuteVz(CLK := stMotionStageVz.bExecute);

fbRealActPositionVec3.x := stMotionStageRx.Axis.NcToPlc.ActPos;
fbRealActPositionVec3.y := stMotionStageRy.Axis.NcToPlc.ActPos;
fbRealActPositionVec3.z := stMotionStageRz.Axis.NcToPlc.ActPos;

fbRealActVelocityVec3.x := stMotionStageRx.Axis.NcToPlc.ActVelo;
fbRealActVelocityVec3.y := stMotionStageRy.Axis.NcToPlc.ActVelo;
fbRealActVelocityVec3.z := stMotionStageRz.Axis.NcToPlc.ActVelo;

fbRealActAcceleraVec3.x := stMotionStageRx.Axis.NcToPlc.ActAcc;
fbRealActAcceleraVec3.y := stMotionStageRy.Axis.NcToPlc.ActAcc;
fbRealActAcceleraVec3.z := stMotionStageRz.Axis.NcToPlc.ActAcc;

sOrderReversed := ReverseOrder(sOrder);

IF bBaseToNew THEN
    RotatePosVelAccFrame(
        fbBaseFramePositionVec3 := fbRealActPositionVec3,
        fbBaseFrameVelocityVec3 := fbRealActVelocityVec3,
        fbBaseFrameAcceleraVec3 := fbRealActAcceleraVec3,
        fbNewFramePositionVec3 => fbVirtActPositionVec3,
        fbNewFrameVelocityVec3 => fbVirtActVelocityVec3,
        fbNewFrameAcceleraVec3 => fbVirtActAcceleraVec3,
        fAlphaRadians := fAlphaRadians,
        fBetaRadians := fBetaRadians,
        fGammaRadians := fGammaRadians,
        sOrder := sOrder
    );
ELSE
    RotatePosVelAccFrame(
        fbBaseFramePositionVec3 := fbRealActPositionVec3,
        fbBaseFrameVelocityVec3 := fbRealActVelocityVec3,
        fbBaseFrameAcceleraVec3 := fbRealActAcceleraVec3,
        fbNewFramePositionVec3 => fbVirtActPositionVec3,
        fbNewFrameVelocityVec3 => fbVirtActVelocityVec3,
        fbNewFrameAcceleraVec3 => fbVirtActAcceleraVec3,
        fAlphaRadians := -fGammaRadians,
        fBetaRadians := -fBetaRadians,
        fGammaRadians := -fAlphaRadians,
        sOrder := sOrderReversed
    );
END_IF

SetTargetPosVelAcc3D(
    stMotionStageX := stMotionStageVx,
    stMotionStageY := stMotionStageVy,
    stMotionStageZ := stMotionStageVz,
    fbActPosVec3 := fbVirtActPositionVec3,
    fbTarPosVec3 => fbVirtTarPositionVec3,
    fbTarVelVec3 => fbVirtTarVelocityVec3,
    fbTarAccVec3 => fbVirtTarAcceleraVec3
);

IF bBaseToNew THEN
    RotatePosVelAccFrame(
        fbBaseFramePositionVec3 := fbVirtTarPositionVec3,
        fbBaseFrameVelocityVec3 := fbVirtTarVelocityVec3,
        fbBaseFrameAcceleraVec3 := fbVirtTarAcceleraVec3,
        fbNewFramePositionVec3 => fbRealTarPositionVec3,
        fbNewFrameVelocityVec3 => fbRealTarVelocityVec3,
        fbNewFrameAcceleraVec3 => fbRealTarAcceleraVec3,
        fAlphaRadians := -fGammaRadians,
        fBetaRadians := -fBetaRadians,
        fGammaRadians := -fAlphaRadians,
        sOrder := sOrderReversed
    );
ELSE
    RotatePosVelAccFrame(
        fbBaseFramePositionVec3 := fbVirtTarPositionVec3,
        fbBaseFrameVelocityVec3 := fbVirtTarVelocityVec3,
        fbBaseFrameAcceleraVec3 := fbVirtTarAcceleraVec3,
        fbNewFramePositionVec3 => fbRealTarPositionVec3,
        fbNewFrameVelocityVec3 => fbRealTarVelocityVec3,
        fbNewFrameAcceleraVec3 => fbRealTarAcceleraVec3,
        fAlphaRadians := fAlphaRadians,
        fBetaRadians := fBetaRadians,
        fGammaRadians := fGammaRadians,
        sOrder := sOrder
    );
END_IF

IF bEnable THEN
    IF rtExecuteVx.Q OR rtExecuteVy.Q OR rtExecuteVz.Q THEN
        stMotionStageRx.fPosition := fbRealTarPositionVec3.x;
        stMotionStageRy.fPosition := fbRealTarPositionVec3.y;
        stMotionStageRz.fPosition := fbRealTarPositionVec3.z;

        stMotionStageRx.fVelocity := ABS(fbRealTarVelocityVec3.x);
        stMotionStageRy.fVelocity := ABS(fbRealTarVelocityVec3.y);
        stMotionStageRz.fVelocity := ABS(fbRealTarVelocityVec3.z);

        stMotionStageRx.fAcceleration := ABS(fbRealTarAcceleraVec3.x);
        stMotionStageRy.fAcceleration := ABS(fbRealTarAcceleraVec3.y);
        stMotionStageRz.fAcceleration := ABS(fbRealTarAcceleraVec3.z);

        stMotionStageRx.fDeceleration := ABS(fbRealTarAcceleraVec3.x);
        stMotionStageRy.fDeceleration := ABS(fbRealTarAcceleraVec3.y);
        stMotionStageRz.fDeceleration := ABS(fbRealTarAcceleraVec3.z);

        IF stMotionStageRx.fVelocity >= 0.001 THEN
            stMotionStageRx.bMoveCmd := TRUE;
        ELSIF ABS(stMotionStageRx.fPosition - stMotionStageRx.Axis.NcToPlc.ActPos) >
                stMotionStageRx.stAxisParameters.fTargetPosControlRange THEN
            stMotionStageRx.fVelocity := 0.001;
            stMotionStageRx.bMoveCmd := TRUE;
        END_IF

        IF stMotionStageRy.fVelocity >= 0.001 THEN
            stMotionStageRy.bMoveCmd := TRUE;
        ELSIF ABS(stMotionStageRy.fPosition - stMotionStageRy.Axis.NcToPlc.ActPos) >
                stMotionStageRy.stAxisParameters.fTargetPosControlRange THEN
            stMotionStageRy.fVelocity := 0.001;
            stMotionStageRy.bMoveCmd := TRUE;
        END_IF

        IF stMotionStageRz.fVelocity >= 0.001 THEN
            stMotionStageRz.bMoveCmd := TRUE;
        ELSIF ABS(stMotionStageRz.fPosition - stMotionStageRz.Axis.NcToPlc.ActPos) >
                stMotionStageRz.stAxisParameters.fTargetPosControlRange THEN
            stMotionStageRz.fVelocity := 0.001;
            stMotionStageRz.bMoveCmd := TRUE;
        END_IF
    END_IF

    IF stMotionStageRx.bError OR stMotionStageRy.bError OR stMotionStageRz.bError THEN
        stMotionStageVx.bError := TRUE;
        stMotionStageVy.bError := TRUE;
        stMotionStageVz.bError := TRUE;
        stMotionStageVx.sCustomErrorMessage := 'An error occured in one of the real axes. All virtual axes stopped.';
        stMotionStageVy.sCustomErrorMessage := 'An error occured in one of the real axes. All virtual axes stopped.';
        stMotionStageVz.sCustomErrorMessage := 'An error occured in one of the real axes. All virtual axes stopped.';
    END_IF
END_IF


METHOD PUBLIC DegToRad : LREAL
VAR_INPUT
    fDeg : LREAL;
END_VAR

DegToRad := fDeg  / 180.0 * lcls_twincat_math.GVL_Constants.PI;
END_METHOD

METHOD ReverseOrder : STRING
VAR_INPUT
    sOrder : STRING;
END_VAR

IF sOrder = '' THEN
    sOrder := 'ZYX';
END_IF
sLeft := LEFT(sOrder, 1);
sMid := MID(sOrder, 1, 2);
sRight := RIGHT(sOrder, 1);
ReverseOrder := CONCAT(sRight, CONCAT(sMid, sLeft));
END_METHOD


METHOD PUBLIC RotatePosVelAccFrame
VAR_INPUT
    fbBaseFramePositionVec3 : FB_Vec3;
    fbBaseFrameVelocityVec3 : FB_Vec3;
    fbBaseFrameAcceleraVec3 : FB_Vec3;

    fAlphaRadians : LREAL;
    fBetaRadians : LREAL;
    fGammaRadians : LREAL;
    sOrder : STRING;
END_VAR
VAR_OUTPUT
    fbNewFramePositionVec3 : FB_Vec3;
    fbNewFrameVelocityVec3 : FB_Vec3;
    fbNewFrameAcceleraVec3 : FB_Vec3;
END_VAR

fbNewFramePositionVec3 := F_EulerRotateVec3Frame(
    iVec3 := fbBaseFramePositionVec3,
    fAlphaRadians := fAlphaRadians,
    fBetaRadians := fBetaRadians,
    fGammaRadians := fGammaRadians,
    sOrder := sOrder
);

fbNewFrameVelocityVec3 := F_EulerRotateVec3Frame(
    iVec3 := fbBaseFrameVelocityVec3,
    fAlphaRadians := fAlphaRadians,
    fBetaRadians := fBetaRadians,
    fGammaRadians := fGammaRadians,
    sOrder := sOrder
);

fbNewFrameAcceleraVec3 := F_EulerRotateVec3Frame(
    iVec3 := fbBaseFrameAcceleraVec3,
    fAlphaRadians := fAlphaRadians,
    fBetaRadians := fBetaRadians,
    fGammaRadians := fGammaRadians,
    sOrder := sOrder
);
END_METHOD


METHOD PUBLIC SetTargetPosVelAcc1D
VAR_INPUT
    stMotionStage : ST_MotionStage;
    fActPos : LREAL;
END_VAR
VAR_OUTPUT
    fTarPos : LREAL;
    fTarVel : LREAL;
    fTarAcc : LREAL;
END_VAR

IF stMotionStage.bBusy THEN
    fTarPos := stMotionStage.fPosition;
    IF fTarPos >= fActPos THEN
        fTarVel := stMotionStage.fVelocity;
        fTarAcc := stMotionStage.fAcceleration;
    ELSE
        fTarVel := -stMotionStage.fVelocity;
        fTarAcc := -stMotionStage.fAcceleration;
    END_IF
ELSE
    fTarPos := fActPos;
    fTarVel := 0.0;
    fTarAcc := 0.0;
END_IF
END_METHOD


METHOD PUBLIC SetTargetPosVelAcc3D
VAR_INPUT
    stMotionStageX : ST_MotionStage;
    stMotionStageY : ST_MotionStage;
    stMotionStageZ : ST_MotionStage;
    fbActPosVec3 : FB_Vec3;
END_VAR
VAR_OUTPUT
    fbTarPosVec3 : FB_Vec3;
    fbTarVelVec3 : FB_Vec3;
    fbTarAccVec3 : FB_Vec3;
END_VAR
VAR
    fTarPosX : LREAL;
    fTarPosY : LREAL;
    fTarPosZ : LREAL;

    fTarVelX : LREAL;
    fTarVelY : LREAL;
    fTarVelZ : LREAL;

    fTarAccX : LREAL;
    fTarAccY : LREAL;
    fTarAccZ : LREAL;
END_VAR

SetTargetPosVelAcc1D(
    stMotionStage := stMotionStageX,
    fActPos := fbActPosVec3.x,
    fTarPos => fTarPosX,
    fTarVel => fTarVelX,
    fTarAcc => fTarAccX
);

SetTargetPosVelAcc1D(
    stMotionStage := stMotionStageY,
    fActPos := fbActPosVec3.y,
    fTarPos => fTarPosY,
    fTarVel => fTarVelY,
    fTarAcc => fTarAccY
);

SetTargetPosVelAcc1D(
    stMotionStage := stMotionStageZ,
    fActPos := fbActPosVec3.z,
    fTarPos => fTarPosZ,
    fTarVel => fTarVelZ,
    fTarAcc => fTarAccZ
);

fbTarPosVec3.Set(fTarPosX, fTarPosY, fTarPosZ);
fbTarVelVec3.Set(fTarVelX, fTarVelY, fTarVelZ);
fbTarAccVec3.Set(fTarAccX, fTarAccY, fTarAccZ);
END_METHOD

END_FUNCTION_BLOCK

// POUs/MotorTesting/FB_MicroStepCountTest
FUNCTION_BLOCK FB_MicroStepCountTest
VAR_INPUT
    bExecute: BOOL;
    fStepSize: LREAL;
    nSteps: UINT;
    fMicroStep: LREAL;
    fVelocity: LREAL;
    tSettleTime: TIME;
END_VAR
VAR_IN_OUT
    Axis: AXIS_REF;
END_VAR
VAR_OUTPUT
    nStepsCounted: UINT;
    nTheorySteps: UINT;
    fPercent: LREAL;
    fEstMicroSize: LREAL;
END_VAR
VAR
    fbMoveRel: MC_MoveRelative;
    fbSettleTimer: TON;
    bDoMove: BOOL;
    nStepCounter: UINT;

    arrPosBuffer: ARRAY [0..99] OF LREAL;
    fAvgPos: LREAL;
    nArrIndex: UINT;
    nLoopIndex: UINT;

    fStartPos: LREAL;
    fPrevPos: LREAL;
    fStepChange: LREAL;

    fStepSum: LREAL;
END_VAR

// Motion FB
fbMoveRel(Axis:=Axis,
    Execute:=bDoMove,
    Distance:=fStepSize,
    Velocity:=fVelocity);

// Settle time
fbSettleTimer(IN:=fbMoveRel.Done,
    PT:=tSettleTime);

// Re-enable the move for next cycle
bDoMove := bExecute AND nStepCounter < nSteps;

// Calculate rolling average
arrPosBuffer[nArrIndex] := Axis.NcToPlc.ActPos;
fAvgPos := 0;
FOR nLoopIndex := 0 TO 99 DO
    fAvgPos := fAvgPos + arrPosBuffer[nLoopIndex];
END_FOR;
fAvgPos := fAvgPos / 100;
nArrIndex := (nArrIndex + 1) MOD 100;

// Initialize starting variables
IF NOT bExecute THEN
    fStartPos := fAvgPos;
    fPrevPos := fAvgPos;
END_IF

// Check results
IF fbSettleTimer.Q THEN
    fStepChange := fAvgPos - fPrevPos;
    // Invert fStepChange if we were doing negative steps
    IF fStepSize < 0 THEN
        fStepChange := fStepChange * -1;
    END_IF
    IF fStepChange > fMicroStep * 0.5 THEN
        nStepsCounted := nStepsCounted + 1;
        fStepSum := fStepSum + fStepChange;
        fEstMicroSize := fStepSum / nStepsCounted;
    END_IF
    nTheorySteps := DINT_TO_UINT(TRUNC(ABS((fStartPos - fAvgPos) / fMicroStep)));
    IF nTheorySteps > 0 THEN
        fPercent := 100 * nStepsCounted / nTheorySteps;
    END_IF
    fPrevPos := fAvgPos;
    nStepCounter := nStepCounter + 1;
    // Reset the move block
    bDoMove := FALSE;
END_IF

END_FUNCTION_BLOCK

// tc_mca_std_lib/POUs/ErrorHandling/FB_ErrorList
FUNCTION_BLOCK FB_ErrorList

VAR_INPUT
	En : BOOL;											//Enable input
	bReset : BOOL;										//Delete all Error entry
	lErrorID : ULINT;									//ErrorID to be acknoledged
	bACK : BOOL;										//Acknoledge the given error and delete it from the list
END_VAR
	
VAR_OUTPUT
	EnO : BOOL;											//Enable output
	nNoError: UINT;										//Number of Errors
	nNoOverflow : INT;									//Number of Overflows
	pErrorSystem : POINTER TO ST_ErrorSystem;			//Pointer to ErrorSystem
END_VAR

VAR
	nFreePos : UINT;									//Number of free position in the list
	nListCnt1 : UINT;									//work variable
	ErrorSystem : ST_ErrorSystem;						//Data structure of the Error list
END_VAR

(*
* ================================================================================
*                                   DESCRIPTION
* ================================================================================
* This Function Block implements the core structure of the Error/Warning Handling
* system. It realizes the datastructure containing every Error Entry, collect
* statistics about the usage and manage the Error Entries.
* Note: The system is under development, most of the functionalities are not
* implemented or existing functionalities may change with time.
* ================================================================================
*)
EnO := En;

//Ponter to ErrorSystem
pErrorSystem := ADR(ErrorSystem);

//Number of overflows
nNoOverflow := ErrorSystem.nNoOverflows;

IF bReset THEN
	MEMSET ( ADR(ErrorSystem.aErrorData[0]), 0, GVL_ErrorSystem.cSizeOfErrorData * SIZEOF(DUT_TerminalError));
	ErrorSystem.lNextErrorID := 1;
END_IF

//Number of errors in the system
nNoError := 0;
FOR nListCnt1 := 0 TO GVL_ErrorSystem.cSizeOfErrorData - 1 DO
	IF ErrorSystem.aErrorData[nListCnt1].Error_ID <> 0  THEN
		nNoError := nNoError+1; 
	END_IF
END_FOR
ErrorSystem.nNoErrors := nNoError;

//Number of free position in the list
nFreePos := GVL_ErrorSystem.cSizeOfErrorData - nNoError;

//Acknoledge specified Error entry
IF bACK THEN
	FOR nListCnt1 := 0 TO GVL_ErrorSystem.cSizeOfErrorData - 1 DO
		IF ErrorSystem.aErrorData[nListCnt1].Error_ID = lErrorID THEN
			ErrorSystem.aErrorData[nListCnt1].ErrorState := DUT_ErrorState.Acknowledged;
		END_IF
	END_FOR
END_IF

//Deleting acknoledged errors
FOR nListCnt1 := 0 TO GVL_ErrorSystem.cSizeOfErrorData - 1 DO
	IF ErrorSystem.aErrorData[nListCnt1].ErrorState = DUT_ErrorState.Acknowledged THEN
		MEMMOVE (ADR(ErrorSystem.aErrorData[nListCnt1]), ADR(ErrorSystem.aErrorData[nListCnt1+1]), (GVL_ErrorSystem.cSizeOfErrorData - 1 - nListCnt1) * SIZEOF(DUT_TerminalError));
		MEMSET(ADR(ErrorSystem.aErrorData[GVL_ErrorSystem.cSizeOfErrorData - 1]), 0, SIZEOF(DUT_TerminalError));
	END_IF
END_FOR

END_FUNCTION_BLOCK

// tc_mca_std_lib/POUs/ErrorHandling/FB_TerminalError
FUNCTION_BLOCK FB_TerminalError

